// TIA Portal project "Project-Sticle" (V15.1)

(* hardware
DEVICE "S71500/ET200MP station_1"  S7-1500 station
   slot 0: "Rail_0"  Rack  6ES7 590-1***0-0AA0
   slot 1: "PLC_1"  CPU 1513-1 PN  6ES7 513-1AL02-0AB0  V2.6
      slot 3: "CPU display_1"  6ES7591-1AA00-0AA0
DEVICE "HMI_1"  KTP900 Basic PN
   slot 0: "HMI_1"  KTP900 Basic PN  6AV2 123-2JB03-0AX0  15.1.0.0
   slot 1: "HMI_RT_1"  KTP900 Basic PN  6AV2 123-2JB03-0AX0  15.1.0.0
   slot 5: "HMI_1.IE_CP_1"  PROFINET Interface  15.0.1.0
      slot 1: "PROFINET Interface_1"  PROFINET Interface
         slot 1: "Port_1"  Port
*)

// ===== PLC "PLC_1"  CPU 1513-1 PN =====

VAR_GLOBAL   // PLC tag table "Default tag table"
   "Clock_Byte" AT %MB0 : Byte;
   "Clock_10Hz" AT %M0.0 : Bool;
   "Clock_5Hz" AT %M0.1 : Bool;
   "Clock_2.5Hz" AT %M0.2 : Bool;
   "Clock_2Hz" AT %M0.3 : Bool;
   "Clock_1.25Hz" AT %M0.4 : Bool;
   "Clock_1Hz" AT %M0.5 : Bool;
   "Clock_0.625Hz" AT %M0.6 : Bool;
   "Clock_0.5Hz" AT %M0.7 : Bool;
END_VAR

DATA_BLOCK "Avarii"   // DB1
{ S7_Optimized_Access := 'TRUE' }
VERSION : 0.1
   VAR
      esd : Bool;
      esd_btn : Bool;
      reset_esd : Bool;
      confirmare_neprimita_actuator : Bool;
      reset_avarii : Bool;
      avarie_imbuteliere : Bool;
      avarie_capace : Bool;
      avarie_eticheta : Bool;
      avarie_impachetare : Bool;
      avarie_cuptor : Bool;
      avarie_generala : Bool;
      timer_confirmare : Time;
      timer_umplere : Time;
      timer_eticheta : Time;
      timer_capac : Time;
      timer_impachetare : Time;
      var_confirmare : Bool;
      timer_secunde_imbuteliere : Time;
      timer_secunde_confirmare : Time;
      timer_secunde_capac : Time;
      timer_secunde_impachetare : Time;
      timer_secunde_eticheta : Time;
      timer_cuptor : Time;
      timer_secunde_cutor : Time;
   END_VAR
BEGIN
END_DATA_BLOCK

DATA_BLOCK "Alarme"   // DB2
{ S7_Optimized_Access := 'TRUE' }
VERSION : 0.1
   VAR
      alarme_gather : Word;
      alarme_vect : Array[0..15] of Bool;
   END_VAR
BEGIN
END_DATA_BLOCK

DATA_BLOCK "Banda"   // DB4
{ S7_Optimized_Access := 'TRUE' }
VERSION : 0.1
   VAR
      banda_pornita_1 : Bool;
      prm_pornire_banda11 : Bool;
      prm_pornire_banda12 : Bool;
      banda_oprita_2 : Bool;
      banda_oprita_3 : Bool;
      banda_oprita_4 : Bool;
      banda_oprita_5 : Bool;
   END_VAR
BEGIN
END_DATA_BLOCK

DATA_BLOCK "Aparate"   // DB5
{ S7_Optimized_Access := 'TRUE' }
VERSION : 0.1
   VAR
      numar_sticle_cerut : UInt;
      numar_sticle_cerut_aux : UInt;
      numar_sticle : UInt;
      inchidere_actuator : Bool;
      deschidere_actuator : Bool;
      confirmare_actuator : Bool;
      timp_umplere_user : Time;
      timp_umplere_secunde : Time;
      terminat_imbuteliere : Bool;
      ajuns_capace : Bool;
      plecat_capace : Bool;
      ajuns_eticheta : Bool;
      plecat_ethicheta : Bool;
      ajuns_impachetare : Bool;
      plecat_impachetare : Bool;
      ajuns_cuptor : Bool;
      plecat_cuptor : Bool;
      nivel_palet : UInt;
      limita_palet : UInt;
      timp_cuptor : Time;
      timp_cuptor_secunde : Time;
   END_VAR
BEGIN
END_DATA_BLOCK

DATA_BLOCK "Butoane/Permisiuni"   // DB6
{ S7_Optimized_Access := 'TRUE' }
VERSION : 0.1
   VAR
      btn_start : Bool;
      permisiune_start : Bool;
      nr_sticle_complet : Bool;
      pauza : Bool;
   END_VAR
BEGIN
END_DATA_BLOCK

DATA_BLOCK "Rising_edges"   // DB7
{ S7_Optimized_Access := 'TRUE' }
VERSION : 0.1
   VAR
      re1 : Bool;
      re2 : Bool;
      re3 : Bool;
      re4 : Bool;
   END_VAR
BEGIN
END_DATA_BLOCK

DATA_BLOCK "Hysteresis_DB"   // DB15
{ S7_Optimized_Access := 'TRUE' }
VERSION : 0.1
// stored: InstanceOfName Hysteresis
"Hysteresis"
BEGIN
END_DATA_BLOCK

DATA_BLOCK "Variabile_Hysteresis"   // DB16
{ S7_Optimized_Access := 'TRUE' }
VERSION : 0.1
   VAR
      bool_cond : Bool;
      Hy_val : Real;
      Setpoint : Real;
      temp : Real;
      lim_inf : Real;
      lim_sup : Real;
      limita_inf_pt_timer : Real;
      dif_lim_inf : Real;
   END_VAR
BEGIN
END_DATA_BLOCK

DATA_BLOCK "Turn_vizual"   // DB17
{ S7_Optimized_Access := 'TRUE' }
VERSION : 0.1
   VAR
      led_rosu : Bool;
      led_verde : Bool;
      led_galben : Bool;
   END_VAR
BEGIN
END_DATA_BLOCK

DATA_BLOCK "Brat_descarcare_DB"   // DB18
{ S7_Optimized_Access := 'TRUE' }
VERSION : 0.1
// stored: InstanceOfName Brat_descarcare
"Brat_descarcare"
BEGIN
END_DATA_BLOCK

DATA_BLOCK "Stari_brat_descarcare"   // DB19
{ S7_Optimized_Access := 'TRUE' }
VERSION : 0.1
   VAR
      ready : Bool;
      finish : Bool;
      running : Bool;
   END_VAR
BEGIN
END_DATA_BLOCK

DATA_BLOCK "Cuastom 0,2HZ clock_DB"   // DB20
{ S7_Optimized_Access := 'TRUE' }
VERSION : 0.1
// stored: InstanceOfName Custom 0,2HZ clock
"Custom 0,2HZ clock"
BEGIN
END_DATA_BLOCK

DATA_BLOCK "Cuptor_DB"   // DB21
{ S7_Optimized_Access := 'TRUE' }
VERSION : 0.1
// stored: InstanceOfName Cuptor
"Cuptor"
BEGIN
END_DATA_BLOCK

// folder: System blocks/Program resources

DATA_BLOCK "timer_confirmare_actuator"   // DB8
{ S7_Optimized_Access := 'TRUE' }
AUTHOR : Simatic
FAMILY : IEC
NAME : IEC_TMR
VERSION : 1.0
// stored: InstanceOfName IEC_TIMER
"IEC_TIMER"
BEGIN
END_DATA_BLOCK

DATA_BLOCK "timer_imbuteliere"   // DB9
{ S7_Optimized_Access := 'TRUE' }
AUTHOR : Simatic
FAMILY : IEC
NAME : IEC_TMR
VERSION : 1.0
// stored: InstanceOfName IEC_TIMER
"IEC_TIMER"
BEGIN
END_DATA_BLOCK

DATA_BLOCK "timer_reset_btn_avarii"   // DB10
{ S7_Optimized_Access := 'TRUE' }
AUTHOR : Simatic
FAMILY : IEC
NAME : IEC_TMR
VERSION : 1.0
// stored: InstanceOfName IEC_TIMER
"IEC_TIMER"
BEGIN
END_DATA_BLOCK

DATA_BLOCK "timer_capace"   // DB11
{ S7_Optimized_Access := 'TRUE' }
AUTHOR : Simatic
FAMILY : IEC
NAME : IEC_TMR
VERSION : 1.0
// stored: InstanceOfName IEC_TIMER
"IEC_TIMER"
BEGIN
END_DATA_BLOCK

DATA_BLOCK "timer_eticheta"   // DB12
{ S7_Optimized_Access := 'TRUE' }
AUTHOR : Simatic
FAMILY : IEC
NAME : IEC_TMR
VERSION : 1.0
// stored: InstanceOfName IEC_TIMER
"IEC_TIMER"
BEGIN
END_DATA_BLOCK

DATA_BLOCK "timer_impachetare"   // DB13
{ S7_Optimized_Access := 'TRUE' }
AUTHOR : Simatic
FAMILY : IEC
NAME : IEC_TMR
VERSION : 1.0
// stored: InstanceOfName IEC_TIMER
"IEC_TIMER"
BEGIN
END_DATA_BLOCK

DATA_BLOCK "reset_esd"   // DB14
{ S7_Optimized_Access := 'TRUE' }
AUTHOR : Simatic
FAMILY : IEC
NAME : IEC_TMR
VERSION : 1.0
// stored: InstanceOfName IEC_TIMER
"IEC_TIMER"
BEGIN
END_DATA_BLOCK

// folder: (top level)

FUNCTION_BLOCK "Hysteresis"   // FB1, LAD
{ S7_Optimized_Access := 'TRUE' }
VERSION : 0.1
   VAR_INPUT
      HY_val : Real;
      Setpoint : Real;
   END_VAR
   VAR_OUTPUT
      h_lim_sup : Real;
      h_lim_inf : Real;
      bool_cond : Bool;
   END_VAR
   VAR_IN_OUT
      temp : Real;
   END_VAR
   VAR
      re1 : Bool;
      re2 : Bool;
      urcare : Bool;
   END_VAR
   VAR_TEMP   // added for the SCL form of the ladder/FBD networks
      _w1 : Bool;
   END_VAR
BEGIN

REGION Network 1: daca are comanda de bool, sa creasca
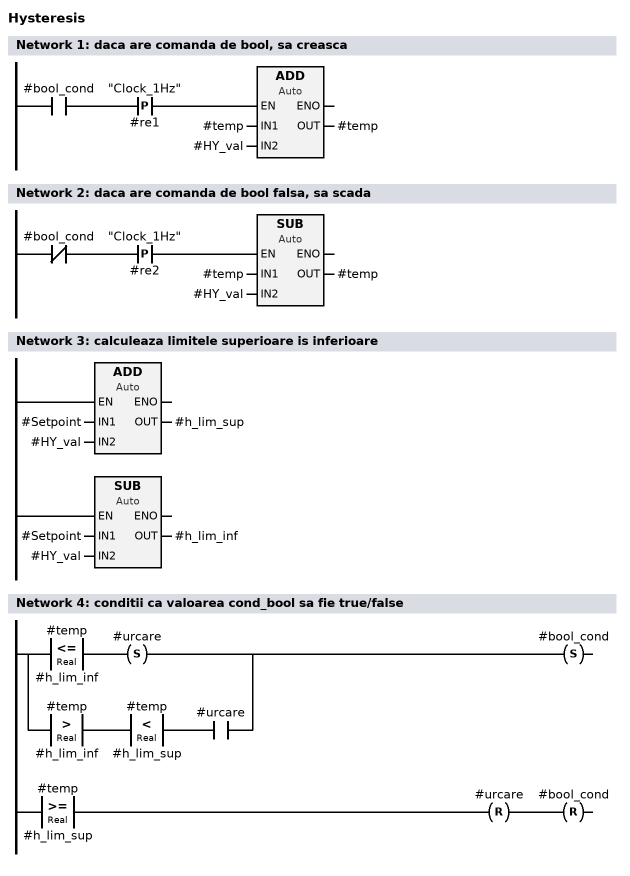
   RUNG wire#powerrail
      Contact( #bool_cond )
      P_Contact(operand := "Clock_1Hz", bit := #re1)
      Add(in1 := #temp, in2 := #HY_val, out => #temp)
   END_RUNG
   // the same network as SCL:
   #_w1 := #bool_cond AND "Clock_1Hz" AND NOT #re1;   // rising edge of "Clock_1Hz"
   #re1 := "Clock_1Hz";
   IF #_w1 THEN #temp := #temp + #HY_val; END_IF;
END_REGION

REGION Network 2: daca are comanda de bool falsa, sa scada
   RUNG wire#powerrail
      I_Contact( #bool_cond )
      P_Contact(operand := "Clock_1Hz", bit := #re2)
      Sub(in1 := #temp, in2 := #HY_val, out => #temp)
   END_RUNG
   // the same network as SCL:
   #_w1 := NOT #bool_cond AND "Clock_1Hz" AND NOT #re2;   // rising edge of "Clock_1Hz"
   #re2 := "Clock_1Hz";
   IF #_w1 THEN #temp := #temp - #HY_val; END_IF;
END_REGION

REGION Network 3: calculeaza limitele superioare is inferioare
   RUNG wire#powerrail
      Add(in1 := #Setpoint, in2 := #HY_val, out => #h_lim_sup)
   END_RUNG
   RUNG wire#powerrail
      Sub(in1 := #Setpoint, in2 := #HY_val, out => #h_lim_inf)
   END_RUNG
   // the same network as SCL:
   #h_lim_sup := #Setpoint + #HY_val;
   #h_lim_inf := #Setpoint - #HY_val;
END_REGION

REGION Network 4: conditii ca valoarea cond_bool sa fie true/false
   RUNG wire#powerrail
      { S7_Templates := "SrcType := Real" } LE_Contact(in1 := #temp, in2 := #h_lim_inf)
      S_Coil( #urcare )
      wire#w1
      S_Coil( #bool_cond )
   END_RUNG
   RUNG wire#powerrail
      { S7_Templates := "SrcType := Real" } GT_Contact(in1 := #temp, in2 := #h_lim_inf)
      { S7_Templates := "SrcType := Real" } LT_Contact(in1 := #temp, in2 := #h_lim_sup)
      Contact( #urcare )
   END_RUNG wire#w1
   RUNG wire#powerrail
      { S7_Templates := "SrcType := Real" } GE_Contact(in1 := #temp, in2 := #h_lim_sup)
      R_Coil( #urcare )
      R_Coil( #bool_cond )
   END_RUNG
   // the same network as SCL:
   #_w1 := #temp <= #h_lim_inf;
   IF #_w1 THEN #urcare := TRUE; END_IF;
   IF #_w1 OR ((#temp > #h_lim_inf) AND (#temp < #h_lim_sup) AND #urcare) THEN #bool_cond := TRUE; END_IF;
   IF #temp >= #h_lim_sup THEN
       #urcare := FALSE;
       #bool_cond := FALSE;
   END_IF;
END_REGION
END_FUNCTION_BLOCK

FUNCTION_BLOCK "Brat_descarcare"   // FB2, LAD
{ S7_Optimized_Access := 'TRUE' }
VERSION : 0.1
   VAR_OUTPUT
      ready : Bool;
      finish : Bool;
      running : Bool;
   END_VAR
   VAR_IN_OUT
      permisiune : Bool;
      nivel_palet : UInt;
   END_VAR
   VAR
      re1 : Bool;
      counter_custom_clock : UInt;
      "bool value" : Bool;
   END_VAR
   VAR_TEMP   // added for the SCL form of the ladder/FBD networks
      _w1 : Bool;
   END_VAR
BEGIN

REGION Network 1: daca e ready si are permisiune, sa treaca pe run
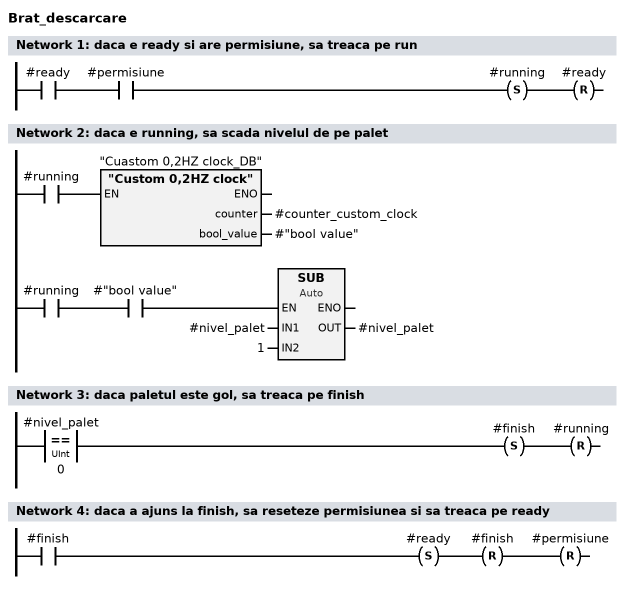
   RUNG wire#powerrail
      Contact( #ready )
      Contact( #permisiune )
      S_Coil( #running )
      R_Coil( #ready )
   END_RUNG
   // the same network as SCL:
   IF #ready AND #permisiune THEN
       #running := TRUE;
       #ready := FALSE;
   END_IF;
END_REGION

REGION Network 2: daca e running, sa scada nivelul de pe palet
   RUNG wire#powerrail
      Contact( #running )
      "Cuastom 0,2HZ clock_DB"("counter" => #counter_custom_clock, bool_value => #"bool value")
   END_RUNG
   RUNG wire#powerrail
      Contact( #running )
      Contact( #"bool value" )
      Sub(in1 := #nivel_palet, in2 := 1, out => #nivel_palet)
   END_RUNG
   // the same network as SCL:
   IF #running THEN
       "Cuastom 0,2HZ clock_DB"("counter" => #counter_custom_clock, bool_value => #"bool value");   // "Custom 0,2HZ clock"
   END_IF;
   IF #running AND #"bool value" THEN #nivel_palet := #nivel_palet - 1; END_IF;
END_REGION

REGION Network 3: daca paletul este gol, sa treaca pe finish
   RUNG wire#powerrail
      { S7_Templates := "SrcType := UInt" } EQ_Contact(in1 := #nivel_palet, in2 := 0)
      S_Coil( #finish )
      R_Coil( #running )
   END_RUNG
   // the same network as SCL:
   IF #nivel_palet = 0 THEN
       #finish := TRUE;
       #running := FALSE;
   END_IF;
END_REGION

REGION Network 4: daca a ajuns la finish, sa reseteze permisiunea si sa treaca pe ready
   RUNG wire#powerrail
      Contact( #finish )
      S_Coil( #ready )
      R_Coil( #finish )
      R_Coil( #permisiune )
   END_RUNG
   // the same network as SCL:
   IF #finish THEN #ready := TRUE; END_IF;
   #_w1 := #finish;
   IF #_w1 THEN
       #finish := FALSE;
       #permisiune := FALSE;
   END_IF;
END_REGION
END_FUNCTION_BLOCK

FUNCTION_BLOCK "Custom 0,2HZ clock"   // FB3, LAD
{ S7_Optimized_Access := 'TRUE' }
VERSION : 0.1
   VAR_OUTPUT
      "counter" : UInt;
      bool_value : Bool;
   END_VAR
   VAR
      re : Bool;
   END_VAR
   VAR_TEMP   // added for the SCL form of the ladder/FBD networks
      _w1 : Bool;
   END_VAR
BEGIN

REGION Network 1: adauga la counter
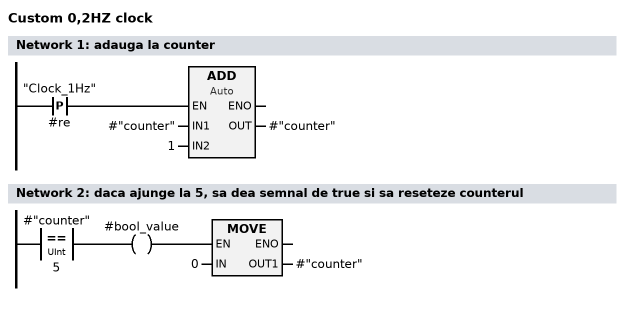
   RUNG wire#powerrail
      P_Contact(operand := "Clock_1Hz", bit := #re)
      Add(in1 := #"counter", in2 := 1, out => #"counter")
   END_RUNG
   // the same network as SCL:
   #_w1 := "Clock_1Hz" AND NOT #re;   // rising edge of "Clock_1Hz"
   #re := "Clock_1Hz";
   IF #_w1 THEN #"counter" := #"counter" + 1; END_IF;
END_REGION

REGION Network 2: daca ajunge la 5, sa dea semnal de true si sa reseteze counterul
   RUNG wire#powerrail
      { S7_Templates := "SrcType := UInt" } EQ_Contact(in1 := #"counter", in2 := 5)
      Coil( #bool_value )
      Move(in := 0, out1 => #"counter")
   END_RUNG
   // the same network as SCL:
   #bool_value := #"counter" = 5;
   IF #bool_value THEN #"counter" := 0; END_IF;
END_REGION
END_FUNCTION_BLOCK

FUNCTION_BLOCK "Cuptor"   // FB4, LAD
{ S7_Optimized_Access := 'TRUE' }
VERSION : 0.1
   VAR_INPUT
      hysteresis_setpoint : Real;
      dif_lim_inf : Real;
      timp_cuptor : Time;
      buton_perm_start : Bool;
      banda_oprita : Bool;
      pauza : Bool;
      avarie_generala : Bool;
      esd : Bool;
   END_VAR
   VAR_OUTPUT
      timer_cuptor_out : Time;
   END_VAR
   VAR_IN_OUT
      b_oprita : Bool;
      plecat_cuptor : Bool;
      ajuns_cuptor : Bool;
      hy_bool_cond : Bool;
      timp_cuptor_sec : Time;
      lim_inf_pt_timer : Real;
      temp : Real;
      hy_val : Real;
      lim_sup : Real;
      lim_inf : Real;
   END_VAR
   VAR
      timer_cuptor : TON_TIME;
   END_VAR
BEGIN

REGION Network 1: calculeaza limita inferioara pt timer la cuptor si timpul in secunde la cuptor
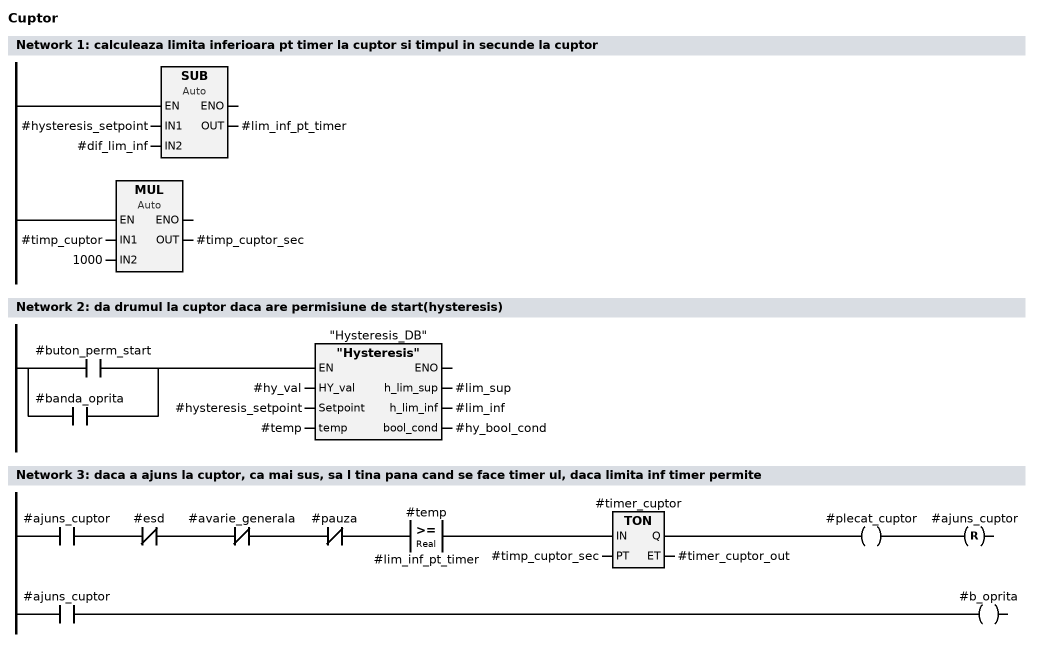
   RUNG wire#powerrail
      Sub(in1 := #hysteresis_setpoint, in2 := #dif_lim_inf, out => #lim_inf_pt_timer)
   END_RUNG
   RUNG wire#powerrail
      Mul(in1 := #timp_cuptor, in2 := 1000, out => #timp_cuptor_sec)
   END_RUNG
   // the same network as SCL:
   #lim_inf_pt_timer := #hysteresis_setpoint - #dif_lim_inf;
   #timp_cuptor_sec := #timp_cuptor * 1000;
END_REGION

REGION Network 2: da drumul la cuptor daca are permisiune de start(hysteresis)
   RUNG wire#powerrail
      Contact( #buton_perm_start )
      wire#w1
      "Hysteresis_DB"(HY_val := #hy_val, Setpoint := #hysteresis_setpoint, temp := #temp, h_lim_sup => #lim_sup, h_lim_inf => #lim_inf, bool_cond => #hy_bool_cond)
   END_RUNG
   RUNG wire#powerrail
      Contact( #banda_oprita )
   END_RUNG wire#w1
   // the same network as SCL:
   IF #buton_perm_start OR #banda_oprita THEN
       "Hysteresis_DB"(HY_val := #hy_val,   // "Hysteresis"
                       Setpoint := #hysteresis_setpoint,
                       temp := #temp,
                       h_lim_sup => #lim_sup,
                       h_lim_inf => #lim_inf,
                       bool_cond => #hy_bool_cond);
   END_IF;
END_REGION

REGION Network 3: daca a ajuns la cuptor, ca mai sus, sa l tina pana cand se face timer ul, daca limita inf timer permite
   #timer_cuptor(IN := #ajuns_cuptor AND NOT #esd AND NOT #avarie_generala AND NOT #pauza AND (#temp >= #lim_inf_pt_timer),   // TON
                 PT := #timp_cuptor_sec,
                 ET => #timer_cuptor_out);
   #plecat_cuptor := #timer_cuptor.Q;
   IF #timer_cuptor.Q THEN #ajuns_cuptor := FALSE; END_IF;
   #b_oprita := #ajuns_cuptor;
END_REGION
END_FUNCTION_BLOCK

ORGANIZATION_BLOCK "Main"   // OB1, LAD, ProgramCycle
TITLE = "Main Program Sweep (Cycle)"
{ S7_Optimized_Access := 'TRUE' }
VERSION : 0.1
   VAR_INPUT
      Initial_Call : Bool;   // Initial call of this OB
      Remanence : Bool;   // =True, if remanent data are available
   END_VAR
   VAR_TEMP   // added for the SCL form of the ladder/FBD networks
      _w1 : Bool;
   END_VAR
BEGIN

REGION Network 1: permisiune start(adauga la final si avarie generala pt fiecare aparat in parte)
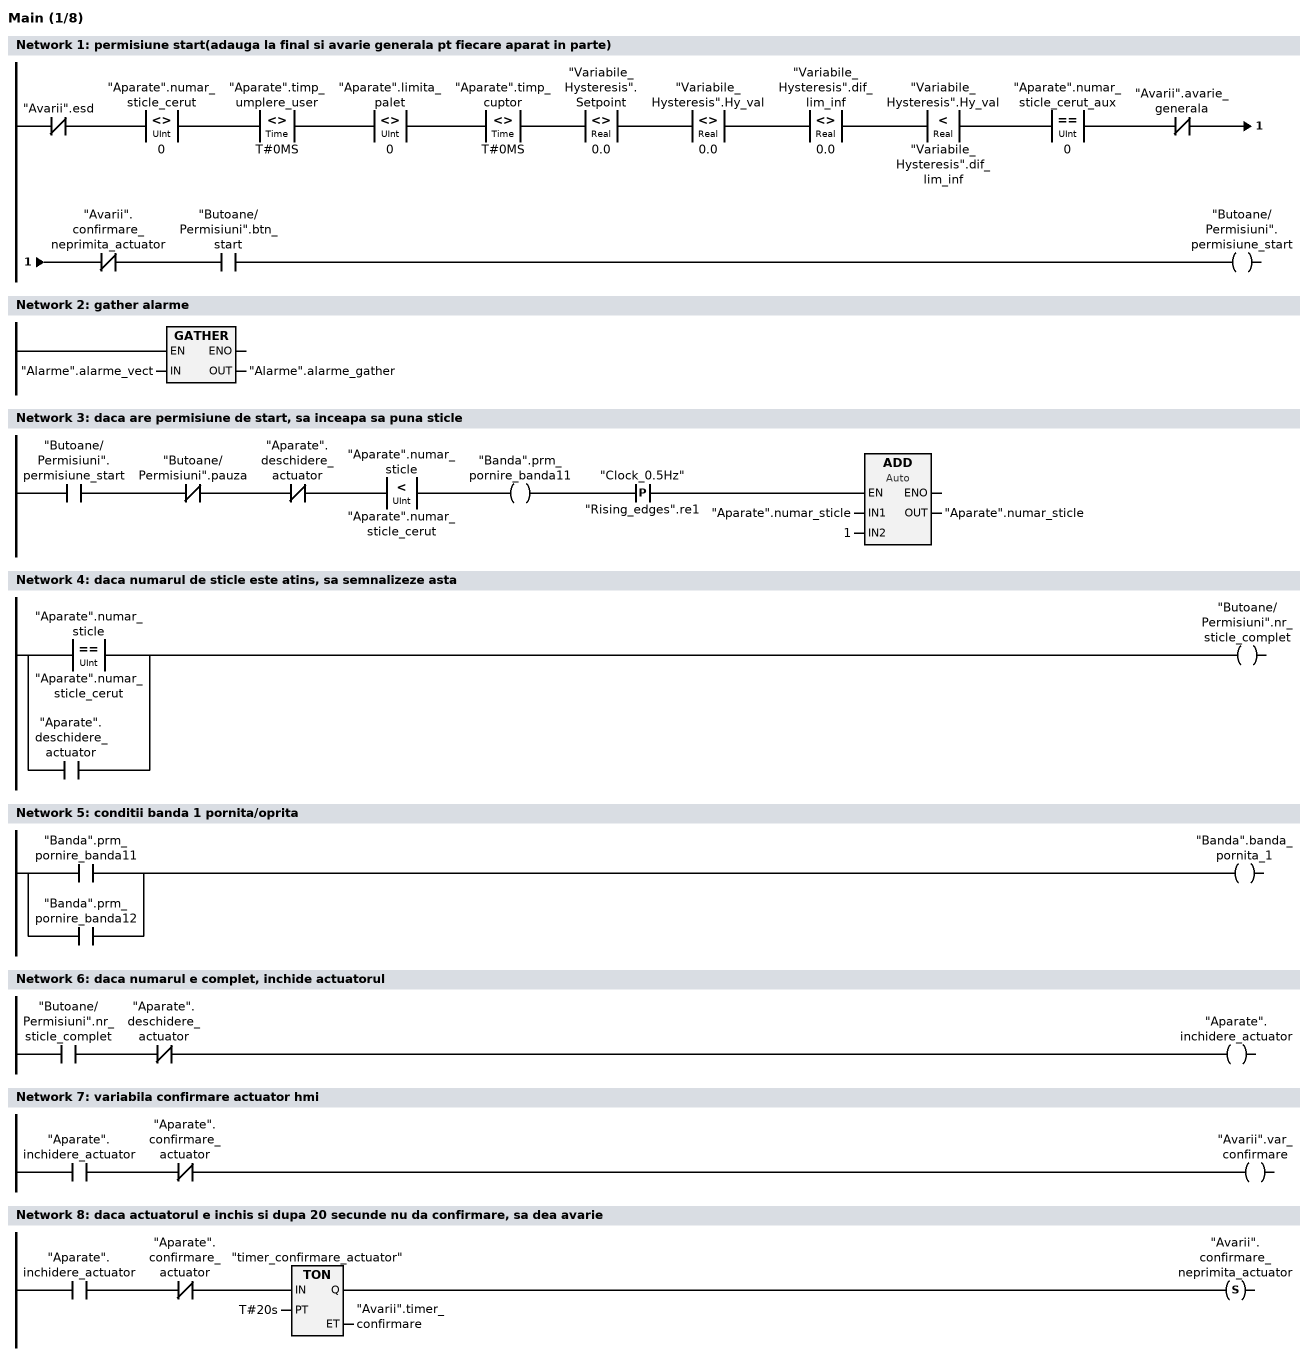
   RUNG wire#powerrail
      I_Contact( "Avarii".esd )
      { S7_Templates := "SrcType := UInt" } NE_Contact(in1 := "Aparate".numar_sticle_cerut, in2 := 0)
      { S7_Templates := "SrcType := Time" } NE_Contact(in1 := "Aparate".timp_umplere_user, in2 := T#0MS)
      { S7_Templates := "SrcType := UInt" } NE_Contact(in1 := "Aparate".limita_palet, in2 := 0)
      { S7_Templates := "SrcType := Time" } NE_Contact(in1 := "Aparate".timp_cuptor, in2 := T#0MS)
      { S7_Templates := "SrcType := Real" } NE_Contact(in1 := "Variabile_Hysteresis".Setpoint, in2 := 0.0)
      { S7_Templates := "SrcType := Real" } NE_Contact(in1 := "Variabile_Hysteresis".Hy_val, in2 := 0.0)
      { S7_Templates := "SrcType := Real" } NE_Contact(in1 := "Variabile_Hysteresis".dif_lim_inf, in2 := 0.0)
      { S7_Templates := "SrcType := Real" } LT_Contact(in1 := "Variabile_Hysteresis".Hy_val, in2 := "Variabile_Hysteresis".dif_lim_inf)
      { S7_Templates := "SrcType := UInt" } EQ_Contact(in1 := "Aparate".numar_sticle_cerut_aux, in2 := 0)
      I_Contact( "Avarii".avarie_generala )
      I_Contact( "Avarii".confirmare_neprimita_actuator )
      Contact( "Butoane/Permisiuni".btn_start )
      Coil( "Butoane/Permisiuni".permisiune_start )
   END_RUNG
   // the same network as SCL:
   "Butoane/Permisiuni".permisiune_start := NOT "Avarii".esd AND ("Aparate".numar_sticle_cerut <> 0) AND ("Aparate".timp_umplere_user <> T#0MS) AND ("Aparate".limita_palet <> 0) AND ("Aparate".timp_cuptor <> T#0MS) AND ("Variabile_Hysteresis".Setpoint <> 0.0) AND ("Variabile_Hysteresis".Hy_val <> 0.0) AND ("Variabile_Hysteresis".dif_lim_inf <> 0.0) AND ("Variabile_Hysteresis".Hy_val < "Variabile_Hysteresis".dif_lim_inf) AND ("Aparate".numar_sticle_cerut_aux = 0) AND NOT "Avarii".avarie_generala AND NOT "Avarii".confirmare_neprimita_actuator AND "Butoane/Permisiuni".btn_start;
END_REGION

REGION Network 2: gather alarme
   GATHER(IN := "Alarme".alarme_vect, OUT => "Alarme".alarme_gather);
END_REGION

REGION Network 3: daca are permisiune de start, sa inceapa sa puna sticle
   RUNG wire#powerrail
      Contact( "Butoane/Permisiuni".permisiune_start )
      I_Contact( "Butoane/Permisiuni".pauza )
      I_Contact( "Aparate".deschidere_actuator )
      { S7_Templates := "SrcType := UInt" } LT_Contact(in1 := "Aparate".numar_sticle, in2 := "Aparate".numar_sticle_cerut)
      Coil( "Banda".prm_pornire_banda11 )
      P_Contact(operand := "Clock_0.5Hz", bit := "Rising_edges".re1)
      Add(in1 := "Aparate".numar_sticle, in2 := 1, out => "Aparate".numar_sticle)
   END_RUNG
   // the same network as SCL:
   "Banda".prm_pornire_banda11 := "Butoane/Permisiuni".permisiune_start AND NOT "Butoane/Permisiuni".pauza AND NOT "Aparate".deschidere_actuator AND ("Aparate".numar_sticle < "Aparate".numar_sticle_cerut);
   #_w1 := "Banda".prm_pornire_banda11 AND "Clock_0.5Hz" AND NOT "Rising_edges".re1;   // rising edge of "Clock_0.5Hz"
   "Rising_edges".re1 := "Clock_0.5Hz";
   IF #_w1 THEN "Aparate".numar_sticle := "Aparate".numar_sticle + 1; END_IF;
END_REGION

REGION Network 4: daca numarul de sticle este atins, sa semnalizeze asta
   RUNG wire#powerrail
      { S7_Templates := "SrcType := UInt" } EQ_Contact(in1 := "Aparate".numar_sticle, in2 := "Aparate".numar_sticle_cerut)
      wire#w1
      Coil( "Butoane/Permisiuni".nr_sticle_complet )
   END_RUNG
   RUNG wire#powerrail
      Contact( "Aparate".deschidere_actuator )
   END_RUNG wire#w1
   // the same network as SCL:
   "Butoane/Permisiuni".nr_sticle_complet := ("Aparate".numar_sticle = "Aparate".numar_sticle_cerut) OR "Aparate".deschidere_actuator;
END_REGION

REGION Network 5: conditii banda 1 pornita/oprita
   RUNG wire#powerrail
      Contact( "Banda".prm_pornire_banda11 )
      wire#w1
      Coil( "Banda".banda_pornita_1 )
   END_RUNG
   RUNG wire#powerrail
      Contact( "Banda".prm_pornire_banda12 )
   END_RUNG wire#w1
   // the same network as SCL:
   "Banda".banda_pornita_1 := "Banda".prm_pornire_banda11 OR "Banda".prm_pornire_banda12;
END_REGION

REGION Network 6: daca numarul e complet, inchide actuatorul
   RUNG wire#powerrail
      Contact( "Butoane/Permisiuni".nr_sticle_complet )
      I_Contact( "Aparate".deschidere_actuator )
      Coil( "Aparate".inchidere_actuator )
   END_RUNG
   // the same network as SCL:
   "Aparate".inchidere_actuator := "Butoane/Permisiuni".nr_sticle_complet AND NOT "Aparate".deschidere_actuator;
END_REGION

REGION Network 7: variabila confirmare actuator hmi
   RUNG wire#powerrail
      Contact( "Aparate".inchidere_actuator )
      I_Contact( "Aparate".confirmare_actuator )
      Coil( "Avarii".var_confirmare )
   END_RUNG
   // the same network as SCL:
   "Avarii".var_confirmare := "Aparate".inchidere_actuator AND NOT "Aparate".confirmare_actuator;
END_REGION

REGION Network 8: daca actuatorul e inchis si dupa 20 secunde nu da confirmare, sa dea avarie
   "timer_confirmare_actuator".TON(IN := "Aparate".inchidere_actuator AND NOT "Aparate".confirmare_actuator,
                           PT := T#20s,
                           ET => "Avarii".timer_confirmare);
   IF "timer_confirmare_actuator".Q THEN "Avarii".confirmare_neprimita_actuator := TRUE; END_IF;
END_REGION

REGION Network 9: daca nr de sticle curent nu este cat cel cerut, sa nu poata sa dea confirmarea actuatorului
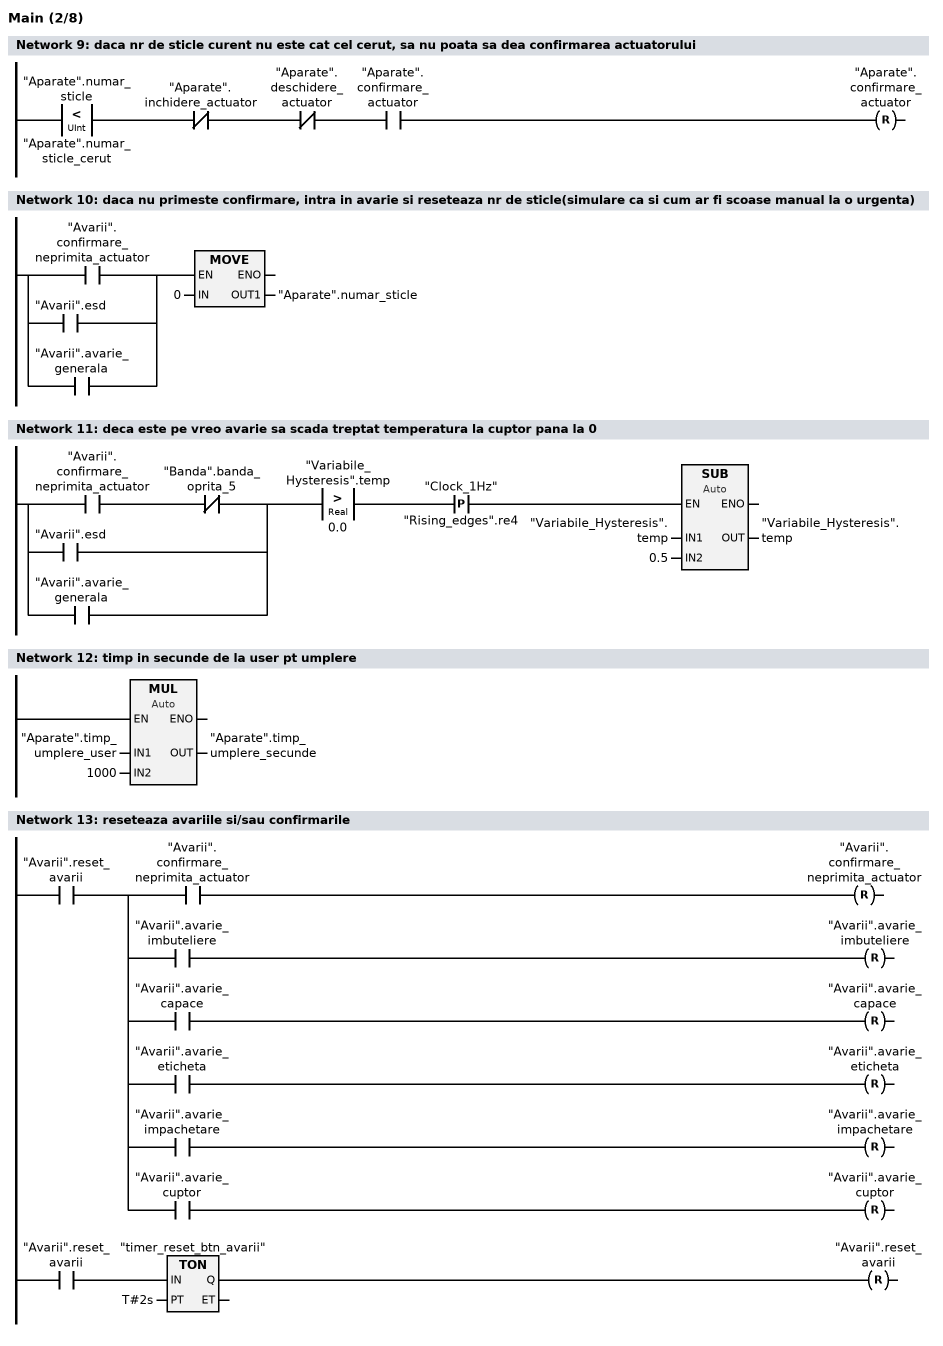
   RUNG wire#powerrail
      { S7_Templates := "SrcType := UInt" } LT_Contact(in1 := "Aparate".numar_sticle, in2 := "Aparate".numar_sticle_cerut)
      I_Contact( "Aparate".inchidere_actuator )
      I_Contact( "Aparate".deschidere_actuator )
      Contact( "Aparate".confirmare_actuator )
      R_Coil( "Aparate".confirmare_actuator )
   END_RUNG
   // the same network as SCL:
   IF ("Aparate".numar_sticle < "Aparate".numar_sticle_cerut) AND NOT "Aparate".inchidere_actuator AND NOT "Aparate".deschidere_actuator AND "Aparate".confirmare_actuator THEN
       "Aparate".confirmare_actuator := FALSE;
   END_IF;
END_REGION

REGION Network 10: daca nu primeste confirmare, intra in avarie si reseteaza nr de sticle(simulare ca si cum ar fi scoase manual la o urgenta)
   RUNG wire#powerrail
      Contact( "Avarii".confirmare_neprimita_actuator )
      wire#w1
      Move(in := 0, out1 => "Aparate".numar_sticle)
   END_RUNG
   RUNG wire#powerrail
      Contact( "Avarii".esd )
   END_RUNG wire#w1
   RUNG wire#powerrail
      Contact( "Avarii".avarie_generala )
   END_RUNG wire#w1
   // the same network as SCL:
   IF "Avarii".confirmare_neprimita_actuator OR "Avarii".esd OR "Avarii".avarie_generala THEN
       "Aparate".numar_sticle := 0;
   END_IF;
END_REGION

REGION Network 11: deca este pe vreo avarie sa scada treptat temperatura la cuptor pana la 0
   RUNG wire#powerrail
      Contact( "Avarii".confirmare_neprimita_actuator )
      I_Contact( "Banda".banda_oprita_5 )
      wire#w1
      { S7_Templates := "SrcType := Real" } GT_Contact(in1 := "Variabile_Hysteresis".temp, in2 := 0.0)
      P_Contact(operand := "Clock_1Hz", bit := "Rising_edges".re4)
      Sub(in1 := "Variabile_Hysteresis".temp, in2 := 0.5, out => "Variabile_Hysteresis".temp)
   END_RUNG
   RUNG wire#powerrail
      Contact( "Avarii".esd )
   END_RUNG wire#w1
   RUNG wire#powerrail
      Contact( "Avarii".avarie_generala )
   END_RUNG wire#w1
   // the same network as SCL:
   #_w1 := (("Avarii".confirmare_neprimita_actuator AND NOT "Banda".banda_oprita_5) OR "Avarii".esd OR "Avarii".avarie_generala) AND ("Variabile_Hysteresis".temp > 0.0) AND "Clock_1Hz" AND NOT "Rising_edges".re4;   // rising edge of "Clock_1Hz"
   "Rising_edges".re4 := "Clock_1Hz";
   IF #_w1 THEN "Variabile_Hysteresis".temp := "Variabile_Hysteresis".temp - 0.5; END_IF;
END_REGION

REGION Network 12: timp in secunde de la user pt umplere
   RUNG wire#powerrail
      Mul(in1 := "Aparate".timp_umplere_user, in2 := 1000, out => "Aparate".timp_umplere_secunde)
   END_RUNG
   // the same network as SCL:
   "Aparate".timp_umplere_secunde := "Aparate".timp_umplere_user * 1000;
END_REGION

REGION Network 13: reseteaza avariile si/sau confirmarile
   IF "Avarii".reset_avarii AND "Avarii".confirmare_neprimita_actuator THEN
       "Avarii".confirmare_neprimita_actuator := FALSE;
   END_IF;
   IF "Avarii".reset_avarii AND "Avarii".avarie_imbuteliere THEN
       "Avarii".avarie_imbuteliere := FALSE;
   END_IF;
   IF "Avarii".reset_avarii AND "Avarii".avarie_capace THEN "Avarii".avarie_capace := FALSE; END_IF;
   IF "Avarii".reset_avarii AND "Avarii".avarie_eticheta THEN "Avarii".avarie_eticheta := FALSE; END_IF;
   IF "Avarii".reset_avarii AND "Avarii".avarie_impachetare THEN
       "Avarii".avarie_impachetare := FALSE;
   END_IF;
   IF "Avarii".reset_avarii AND "Avarii".avarie_cuptor THEN "Avarii".avarie_cuptor := FALSE; END_IF;
   "timer_reset_btn_avarii".TON(IN := "Avarii".reset_avarii, PT := T#2s);
   IF "timer_reset_btn_avarii".Q THEN "Avarii".reset_avarii := FALSE; END_IF;
END_REGION

REGION Network 14: reseteaza butonul de start in caz de esd/avarie
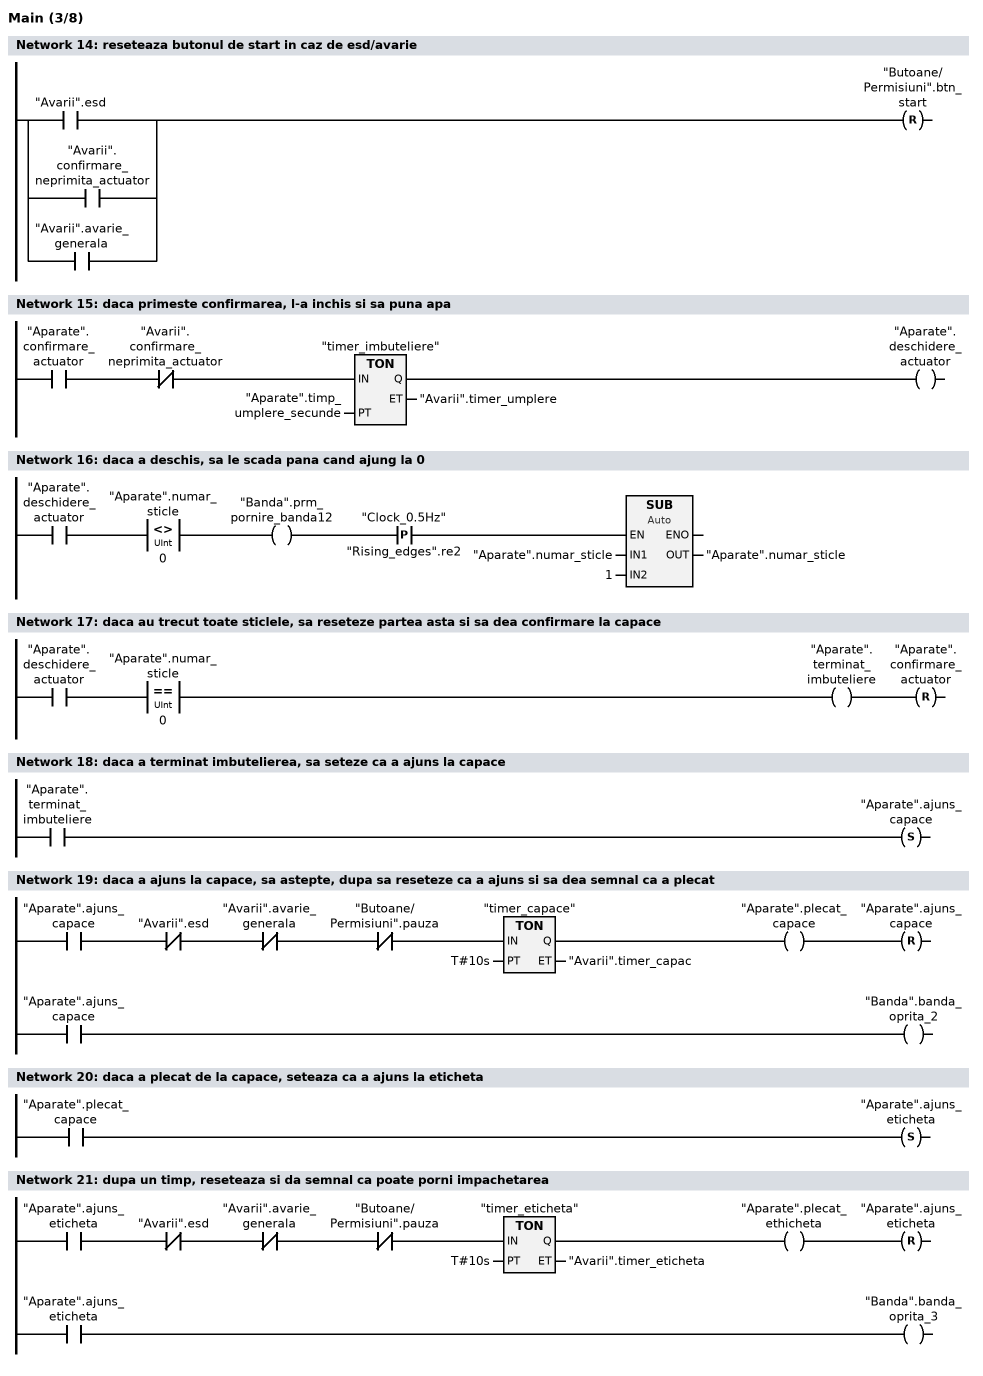
   RUNG wire#powerrail
      Contact( "Avarii".esd )
      wire#w1
      R_Coil( "Butoane/Permisiuni".btn_start )
   END_RUNG
   RUNG wire#powerrail
      Contact( "Avarii".confirmare_neprimita_actuator )
   END_RUNG wire#w1
   RUNG wire#powerrail
      Contact( "Avarii".avarie_generala )
   END_RUNG wire#w1
   // the same network as SCL:
   IF "Avarii".esd OR "Avarii".confirmare_neprimita_actuator OR "Avarii".avarie_generala THEN
       "Butoane/Permisiuni".btn_start := FALSE;
   END_IF;
END_REGION

REGION Network 15: daca primeste confirmarea, l-a inchis si sa puna apa
   "timer_imbuteliere".TON(IN := "Aparate".confirmare_actuator AND NOT "Avarii".confirmare_neprimita_actuator,
                           PT := "Aparate".timp_umplere_secunde,
                           ET => "Avarii".timer_umplere);
   "Aparate".deschidere_actuator := "timer_imbuteliere".Q;
END_REGION

REGION Network 16: daca a deschis, sa le scada pana cand ajung la 0
   RUNG wire#powerrail
      Contact( "Aparate".deschidere_actuator )
      { S7_Templates := "SrcType := UInt" } NE_Contact(in1 := "Aparate".numar_sticle, in2 := 0)
      Coil( "Banda".prm_pornire_banda12 )
      P_Contact(operand := "Clock_0.5Hz", bit := "Rising_edges".re2)
      Sub(in1 := "Aparate".numar_sticle, in2 := 1, out => "Aparate".numar_sticle)
   END_RUNG
   // the same network as SCL:
   "Banda".prm_pornire_banda12 := "Aparate".deschidere_actuator AND ("Aparate".numar_sticle <> 0);
   #_w1 := "Banda".prm_pornire_banda12 AND "Clock_0.5Hz" AND NOT "Rising_edges".re2;   // rising edge of "Clock_0.5Hz"
   "Rising_edges".re2 := "Clock_0.5Hz";
   IF #_w1 THEN "Aparate".numar_sticle := "Aparate".numar_sticle - 1; END_IF;
END_REGION

REGION Network 17: daca au trecut toate sticlele, sa reseteze partea asta si sa dea confirmare la capace
   RUNG wire#powerrail
      Contact( "Aparate".deschidere_actuator )
      { S7_Templates := "SrcType := UInt" } EQ_Contact(in1 := "Aparate".numar_sticle, in2 := 0)
      Coil( "Aparate".terminat_imbuteliere )
      R_Coil( "Aparate".confirmare_actuator )
   END_RUNG
   // the same network as SCL:
   "Aparate".terminat_imbuteliere := "Aparate".deschidere_actuator AND ("Aparate".numar_sticle = 0);
   IF "Aparate".terminat_imbuteliere THEN "Aparate".confirmare_actuator := FALSE; END_IF;
END_REGION

REGION Network 18: daca a terminat imbutelierea, sa seteze ca a ajuns la capace
   RUNG wire#powerrail
      Contact( "Aparate".terminat_imbuteliere )
      S_Coil( "Aparate".ajuns_capace )
   END_RUNG
   // the same network as SCL:
   IF "Aparate".terminat_imbuteliere THEN "Aparate".ajuns_capace := TRUE; END_IF;
END_REGION

REGION Network 19: daca a ajuns la capace, sa astepte, dupa sa reseteze ca a ajuns si sa dea semnal ca a plecat
   "timer_capace".TON(IN := "Aparate".ajuns_capace AND NOT "Avarii".esd AND NOT "Avarii".avarie_generala AND NOT "Butoane/Permisiuni".pauza,
                      PT := T#10s,
                      ET => "Avarii".timer_capac);
   "Aparate".plecat_capace := "timer_capace".Q;
   IF "timer_capace".Q THEN "Aparate".ajuns_capace := FALSE; END_IF;
   "Banda".banda_oprita_2 := "Aparate".ajuns_capace;
END_REGION

REGION Network 20: daca a plecat de la capace, seteaza ca a ajuns la eticheta
   RUNG wire#powerrail
      Contact( "Aparate".plecat_capace )
      S_Coil( "Aparate".ajuns_eticheta )
   END_RUNG
   // the same network as SCL:
   IF "Aparate".plecat_capace THEN "Aparate".ajuns_eticheta := TRUE; END_IF;
END_REGION

REGION Network 21: dupa un timp, reseteaza si da semnal ca poate porni impachetarea
   "timer_eticheta".TON(IN := "Aparate".ajuns_eticheta AND NOT "Avarii".esd AND NOT "Avarii".avarie_generala AND NOT "Butoane/Permisiuni".pauza,
                        PT := T#10s,
                        ET => "Avarii".timer_eticheta);
   "Aparate".plecat_ethicheta := "timer_eticheta".Q;
   IF "timer_eticheta".Q THEN "Aparate".ajuns_eticheta := FALSE; END_IF;
   "Banda".banda_oprita_3 := "Aparate".ajuns_eticheta;
END_REGION

REGION Network 22: seteaza ca a ajuns la impachetare
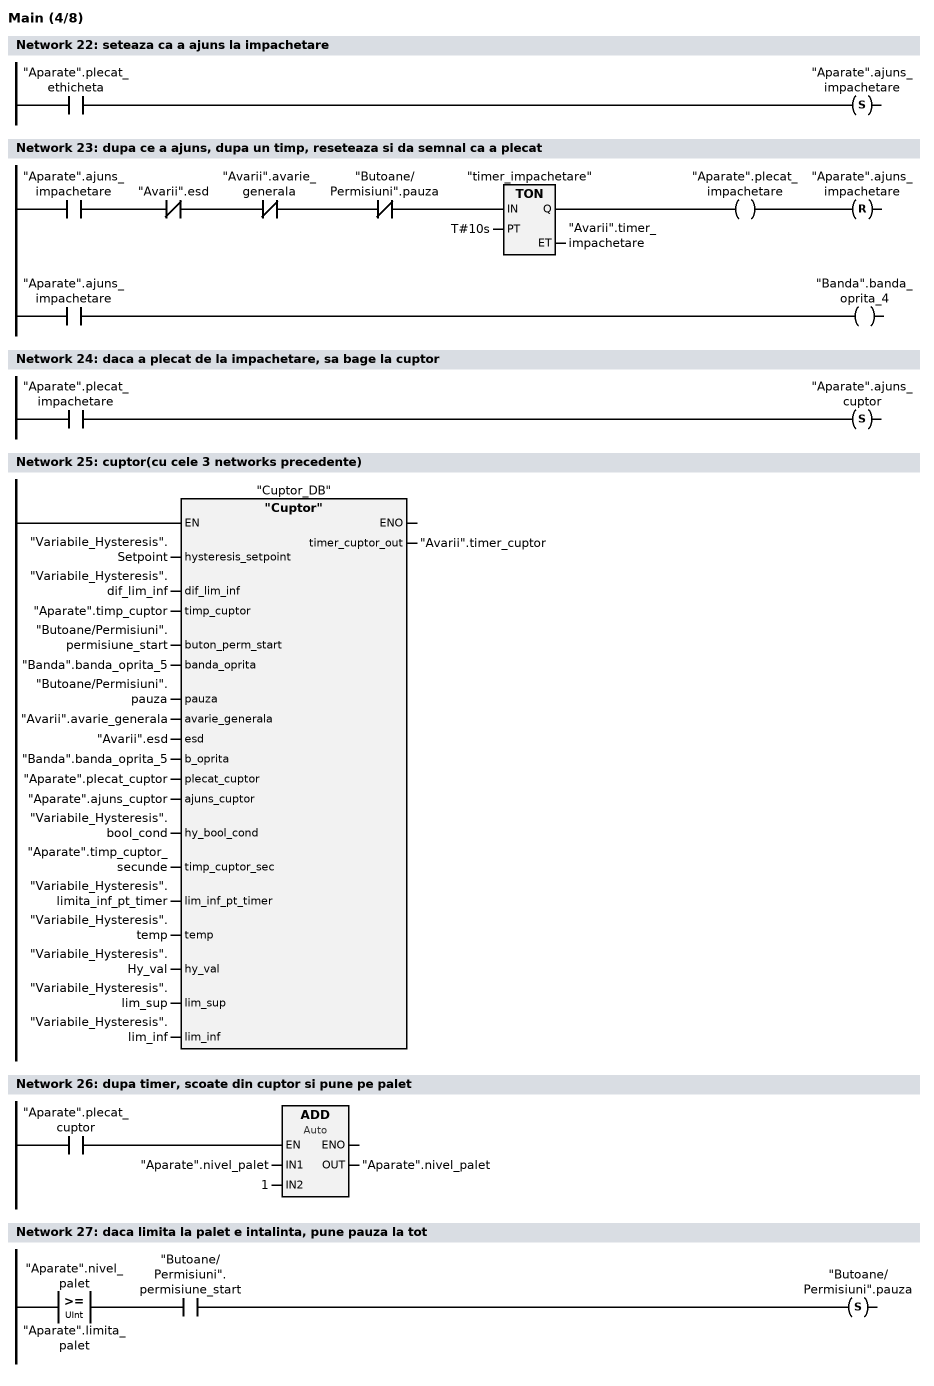
   RUNG wire#powerrail
      Contact( "Aparate".plecat_ethicheta )
      S_Coil( "Aparate".ajuns_impachetare )
   END_RUNG
   // the same network as SCL:
   IF "Aparate".plecat_ethicheta THEN "Aparate".ajuns_impachetare := TRUE; END_IF;
END_REGION

REGION Network 23: dupa ce a ajuns, dupa un timp, reseteaza si da semnal ca a plecat
   "timer_impachetare".TON(IN := "Aparate".ajuns_impachetare AND NOT "Avarii".esd AND NOT "Avarii".avarie_generala AND NOT "Butoane/Permisiuni".pauza,
                           PT := T#10s,
                           ET => "Avarii".timer_impachetare);
   "Aparate".plecat_impachetare := "timer_impachetare".Q;
   IF "timer_impachetare".Q THEN "Aparate".ajuns_impachetare := FALSE; END_IF;
   "Banda".banda_oprita_4 := "Aparate".ajuns_impachetare;
END_REGION

REGION Network 24: daca a plecat de la impachetare, sa bage la cuptor
   RUNG wire#powerrail
      Contact( "Aparate".plecat_impachetare )
      S_Coil( "Aparate".ajuns_cuptor )
   END_RUNG
   // the same network as SCL:
   IF "Aparate".plecat_impachetare THEN "Aparate".ajuns_cuptor := TRUE; END_IF;
END_REGION

REGION Network 25: cuptor(cu cele 3 networks precedente)
   RUNG wire#powerrail
      "Cuptor_DB"(hysteresis_setpoint := "Variabile_Hysteresis".Setpoint, dif_lim_inf := "Variabile_Hysteresis".dif_lim_inf, timp_cuptor := "Aparate".timp_cuptor, buton_perm_start := "Butoane/Permisiuni".permisiune_start, banda_oprita := "Banda".banda_oprita_5, pauza := "Butoane/Permisiuni".pauza, avarie_generala := "Avarii".avarie_generala, esd := "Avarii".esd, b_oprita := "Banda".banda_oprita_5, plecat_cuptor := "Aparate".plecat_cuptor, ajuns_cuptor := "Aparate".ajuns_cuptor, hy_bool_cond := "Variabile_Hysteresis".bool_cond, timp_cuptor_sec := "Aparate".timp_cuptor_secunde, lim_inf_pt_timer := "Variabile_Hysteresis".limita_inf_pt_timer, temp := "Variabile_Hysteresis".temp, hy_val := "Variabile_Hysteresis".Hy_val, lim_sup := "Variabile_Hysteresis".lim_sup, lim_inf := "Variabile_Hysteresis".lim_inf, timer_cuptor_out => "Avarii".timer_cuptor)
   END_RUNG
   // the same network as SCL:
   "Cuptor_DB"(hysteresis_setpoint := "Variabile_Hysteresis".Setpoint,   // "Cuptor"
               dif_lim_inf := "Variabile_Hysteresis".dif_lim_inf,
               timp_cuptor := "Aparate".timp_cuptor,
               buton_perm_start := "Butoane/Permisiuni".permisiune_start,
               banda_oprita := "Banda".banda_oprita_5,
               pauza := "Butoane/Permisiuni".pauza,
               avarie_generala := "Avarii".avarie_generala,
               esd := "Avarii".esd,
               b_oprita := "Banda".banda_oprita_5,
               plecat_cuptor := "Aparate".plecat_cuptor,
               ajuns_cuptor := "Aparate".ajuns_cuptor,
               hy_bool_cond := "Variabile_Hysteresis".bool_cond,
               timp_cuptor_sec := "Aparate".timp_cuptor_secunde,
               lim_inf_pt_timer := "Variabile_Hysteresis".limita_inf_pt_timer,
               temp := "Variabile_Hysteresis".temp,
               hy_val := "Variabile_Hysteresis".Hy_val,
               lim_sup := "Variabile_Hysteresis".lim_sup,
               lim_inf := "Variabile_Hysteresis".lim_inf,
               timer_cuptor_out => "Avarii".timer_cuptor);
END_REGION

REGION Network 26: dupa timer, scoate din cuptor si pune pe palet
   RUNG wire#powerrail
      Contact( "Aparate".plecat_cuptor )
      Add(in1 := "Aparate".nivel_palet, in2 := 1, out => "Aparate".nivel_palet)
   END_RUNG
   // the same network as SCL:
   IF "Aparate".plecat_cuptor THEN "Aparate".nivel_palet := "Aparate".nivel_palet + 1; END_IF;
END_REGION

REGION Network 27: daca limita la palet e intalinta, pune pauza la tot
   RUNG wire#powerrail
      { S7_Templates := "SrcType := UInt" } GE_Contact(in1 := "Aparate".nivel_palet, in2 := "Aparate".limita_palet)
      Contact( "Butoane/Permisiuni".permisiune_start )
      S_Coil( "Butoane/Permisiuni".pauza )
   END_RUNG
   // the same network as SCL:
   IF ("Aparate".nivel_palet >= "Aparate".limita_palet) AND "Butoane/Permisiuni".permisiune_start THEN
       "Butoane/Permisiuni".pauza := TRUE;
   END_IF;
END_REGION

REGION Network 28: simuleaza aici turnul vizual RGV
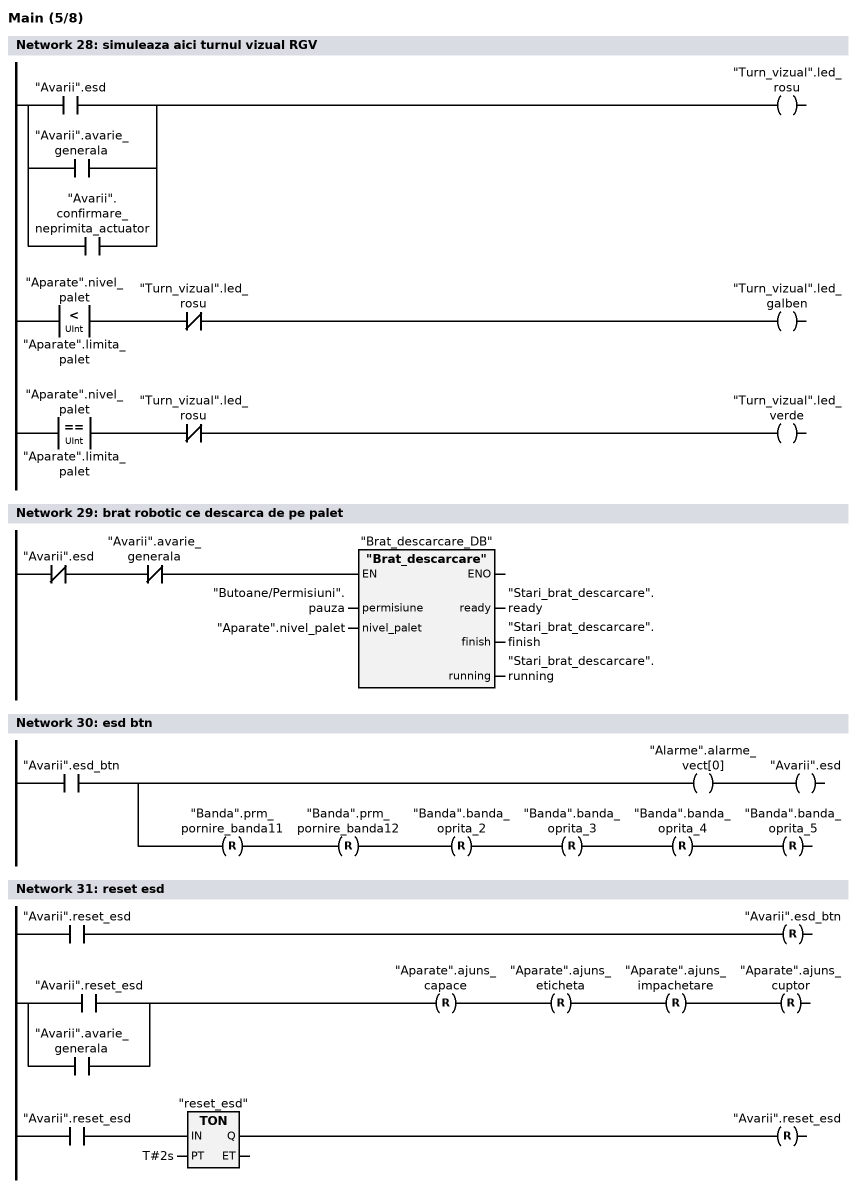
   RUNG wire#powerrail
      Contact( "Avarii".esd )
      wire#w1
      Coil( "Turn_vizual".led_rosu )
   END_RUNG
   RUNG wire#powerrail
      Contact( "Avarii".avarie_generala )
   END_RUNG wire#w1
   RUNG wire#powerrail
      Contact( "Avarii".confirmare_neprimita_actuator )
   END_RUNG wire#w1
   RUNG wire#powerrail
      { S7_Templates := "SrcType := UInt" } LT_Contact(in1 := "Aparate".nivel_palet, in2 := "Aparate".limita_palet)
      I_Contact( "Turn_vizual".led_rosu )
      Coil( "Turn_vizual".led_galben )
   END_RUNG
   RUNG wire#powerrail
      { S7_Templates := "SrcType := UInt" } EQ_Contact(in1 := "Aparate".nivel_palet, in2 := "Aparate".limita_palet)
      I_Contact( "Turn_vizual".led_rosu )
      Coil( "Turn_vizual".led_verde )
   END_RUNG
   // the same network as SCL:
   "Turn_vizual".led_rosu := "Avarii".esd OR "Avarii".avarie_generala OR "Avarii".confirmare_neprimita_actuator;
   "Turn_vizual".led_galben := ("Aparate".nivel_palet < "Aparate".limita_palet) AND NOT "Turn_vizual".led_rosu;
   "Turn_vizual".led_verde := ("Aparate".nivel_palet = "Aparate".limita_palet) AND NOT "Turn_vizual".led_rosu;
END_REGION

REGION Network 29: brat robotic ce descarca de pe palet
   RUNG wire#powerrail
      I_Contact( "Avarii".esd )
      I_Contact( "Avarii".avarie_generala )
      "Brat_descarcare_DB"(permisiune := "Butoane/Permisiuni".pauza, nivel_palet := "Aparate".nivel_palet, ready => "Stari_brat_descarcare".ready, finish => "Stari_brat_descarcare".finish, running => "Stari_brat_descarcare".running)
   END_RUNG
   // the same network as SCL:
   IF NOT "Avarii".esd AND NOT "Avarii".avarie_generala THEN
       "Brat_descarcare_DB"(permisiune := "Butoane/Permisiuni".pauza,   // "Brat_descarcare"
                            nivel_palet := "Aparate".nivel_palet,
                            ready => "Stari_brat_descarcare".ready,
                            finish => "Stari_brat_descarcare".finish,
                            running => "Stari_brat_descarcare".running);
   END_IF;
END_REGION

REGION Network 30: esd btn
   RUNG wire#powerrail
      Contact( "Avarii".esd_btn )
      wire#w1
      Coil( "Alarme".alarme_vect[0] )
      Coil( "Avarii".esd )
   END_RUNG
   RUNG wire#w1
      R_Coil( "Banda".prm_pornire_banda11 )
      R_Coil( "Banda".prm_pornire_banda12 )
      R_Coil( "Banda".banda_oprita_2 )
      R_Coil( "Banda".banda_oprita_3 )
      R_Coil( "Banda".banda_oprita_4 )
      R_Coil( "Banda".banda_oprita_5 )
   END_RUNG
   // the same network as SCL:
   "Alarme".alarme_vect[0] := "Avarii".esd_btn;
   "Avarii".esd := "Avarii".esd_btn;
   IF "Avarii".esd_btn THEN
       "Banda".prm_pornire_banda11 := FALSE;
       "Banda".prm_pornire_banda12 := FALSE;
       "Banda".banda_oprita_2 := FALSE;
       "Banda".banda_oprita_3 := FALSE;
       "Banda".banda_oprita_4 := FALSE;
       "Banda".banda_oprita_5 := FALSE;
   END_IF;
END_REGION

REGION Network 31: reset esd
   IF "Avarii".reset_esd THEN "Avarii".esd_btn := FALSE; END_IF;
   IF "Avarii".reset_esd OR "Avarii".avarie_generala THEN
       "Aparate".ajuns_capace := FALSE;
       "Aparate".ajuns_eticheta := FALSE;
       "Aparate".ajuns_impachetare := FALSE;
       "Aparate".ajuns_cuptor := FALSE;
   END_IF;
   "reset_esd".TON(IN := "Avarii".reset_esd, PT := T#2s);
   IF "reset_esd".Q THEN "Avarii".reset_esd := FALSE; END_IF;
END_REGION

REGION Network 32: avarie generala provocata de o avarie la unul din aparate
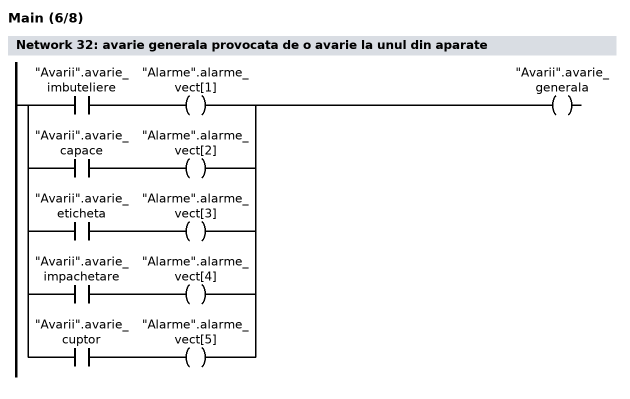
   RUNG wire#powerrail
      Contact( "Avarii".avarie_imbuteliere )
      Coil( "Alarme".alarme_vect[1] )
      wire#w1
      Coil( "Avarii".avarie_generala )
   END_RUNG
   RUNG wire#powerrail
      Contact( "Avarii".avarie_capace )
      Coil( "Alarme".alarme_vect[2] )
   END_RUNG wire#w1
   RUNG wire#powerrail
      Contact( "Avarii".avarie_eticheta )
      Coil( "Alarme".alarme_vect[3] )
   END_RUNG wire#w1
   RUNG wire#powerrail
      Contact( "Avarii".avarie_impachetare )
      Coil( "Alarme".alarme_vect[4] )
   END_RUNG wire#w1
   RUNG wire#powerrail
      Contact( "Avarii".avarie_cuptor )
      Coil( "Alarme".alarme_vect[5] )
   END_RUNG wire#w1
   // the same network as SCL:
   "Alarme".alarme_vect[1] := "Avarii".avarie_imbuteliere;
   "Alarme".alarme_vect[2] := "Avarii".avarie_capace;
   "Alarme".alarme_vect[3] := "Avarii".avarie_eticheta;
   "Alarme".alarme_vect[4] := "Avarii".avarie_impachetare;
   "Alarme".alarme_vect[5] := "Avarii".avarie_cuptor;
   "Avarii".avarie_generala := "Avarii".avarie_imbuteliere OR "Avarii".avarie_capace OR "Avarii".avarie_eticheta OR "Avarii".avarie_impachetare OR "Avarii".avarie_cuptor;
END_REGION

REGION Network 33: setare alarme hmi
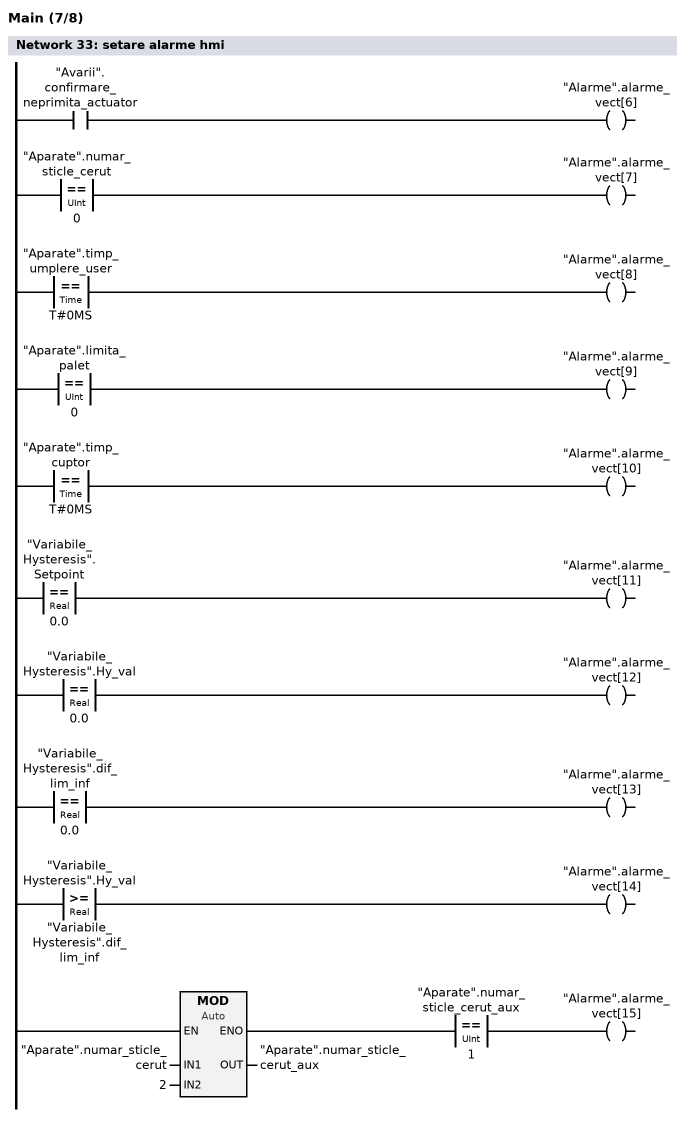
   RUNG wire#powerrail
      Contact( "Avarii".confirmare_neprimita_actuator )
      Coil( "Alarme".alarme_vect[6] )
   END_RUNG
   RUNG wire#powerrail
      { S7_Templates := "SrcType := UInt" } EQ_Contact(in1 := "Aparate".numar_sticle_cerut, in2 := 0)
      Coil( "Alarme".alarme_vect[7] )
   END_RUNG
   RUNG wire#powerrail
      { S7_Templates := "SrcType := Time" } EQ_Contact(in1 := "Aparate".timp_umplere_user, in2 := T#0MS)
      Coil( "Alarme".alarme_vect[8] )
   END_RUNG
   RUNG wire#powerrail
      { S7_Templates := "SrcType := UInt" } EQ_Contact(in1 := "Aparate".limita_palet, in2 := 0)
      Coil( "Alarme".alarme_vect[9] )
   END_RUNG
   RUNG wire#powerrail
      { S7_Templates := "SrcType := Time" } EQ_Contact(in1 := "Aparate".timp_cuptor, in2 := T#0MS)
      Coil( "Alarme".alarme_vect[10] )
   END_RUNG
   RUNG wire#powerrail
      { S7_Templates := "SrcType := Real" } EQ_Contact(in1 := "Variabile_Hysteresis".Setpoint, in2 := 0.0)
      Coil( "Alarme".alarme_vect[11] )
   END_RUNG
   RUNG wire#powerrail
      { S7_Templates := "SrcType := Real" } EQ_Contact(in1 := "Variabile_Hysteresis".Hy_val, in2 := 0.0)
      Coil( "Alarme".alarme_vect[12] )
   END_RUNG
   RUNG wire#powerrail
      { S7_Templates := "SrcType := Real" } EQ_Contact(in1 := "Variabile_Hysteresis".dif_lim_inf, in2 := 0.0)
      Coil( "Alarme".alarme_vect[13] )
   END_RUNG
   RUNG wire#powerrail
      { S7_Templates := "SrcType := Real" } GE_Contact(in1 := "Variabile_Hysteresis".Hy_val, in2 := "Variabile_Hysteresis".dif_lim_inf)
      Coil( "Alarme".alarme_vect[14] )
   END_RUNG
   RUNG wire#powerrail
      Mod(in1 := "Aparate".numar_sticle_cerut, in2 := 2, out => "Aparate".numar_sticle_cerut_aux)
      { S7_Templates := "SrcType := UInt" } EQ_Contact(in1 := "Aparate".numar_sticle_cerut_aux, in2 := 1)
      Coil( "Alarme".alarme_vect[15] )
   END_RUNG
   // the same network as SCL:
   "Alarme".alarme_vect[6] := "Avarii".confirmare_neprimita_actuator;
   "Alarme".alarme_vect[7] := "Aparate".numar_sticle_cerut = 0;
   "Alarme".alarme_vect[8] := "Aparate".timp_umplere_user = T#0MS;
   "Alarme".alarme_vect[9] := "Aparate".limita_palet = 0;
   "Alarme".alarme_vect[10] := "Aparate".timp_cuptor = T#0MS;
   "Alarme".alarme_vect[11] := "Variabile_Hysteresis".Setpoint = 0.0;
   "Alarme".alarme_vect[12] := "Variabile_Hysteresis".Hy_val = 0.0;
   "Alarme".alarme_vect[13] := "Variabile_Hysteresis".dif_lim_inf = 0.0;
   "Alarme".alarme_vect[14] := "Variabile_Hysteresis".Hy_val >= "Variabile_Hysteresis".dif_lim_inf;
   "Aparate".numar_sticle_cerut_aux := "Aparate".numar_sticle_cerut MOD 2;
   "Alarme".alarme_vect[15] := "Aparate".numar_sticle_cerut_aux = 1;
END_REGION

REGION Network 34: timp in secunde pt simulare (pe hmi)
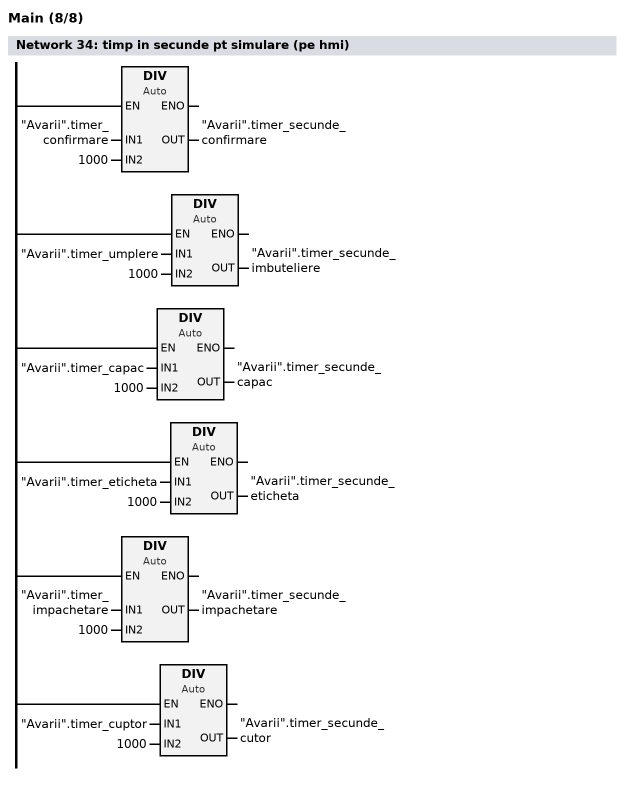
   RUNG wire#powerrail
      Div(in1 := "Avarii".timer_confirmare, in2 := 1000, out => "Avarii".timer_secunde_confirmare)
   END_RUNG
   RUNG wire#powerrail
      Div(in1 := "Avarii".timer_umplere, in2 := 1000, out => "Avarii".timer_secunde_imbuteliere)
   END_RUNG
   RUNG wire#powerrail
      Div(in1 := "Avarii".timer_capac, in2 := 1000, out => "Avarii".timer_secunde_capac)
   END_RUNG
   RUNG wire#powerrail
      Div(in1 := "Avarii".timer_eticheta, in2 := 1000, out => "Avarii".timer_secunde_eticheta)
   END_RUNG
   RUNG wire#powerrail
      Div(in1 := "Avarii".timer_impachetare, in2 := 1000, out => "Avarii".timer_secunde_impachetare)
   END_RUNG
   RUNG wire#powerrail
      Div(in1 := "Avarii".timer_cuptor, in2 := 1000, out => "Avarii".timer_secunde_cutor)
   END_RUNG
   // the same network as SCL:
   "Avarii".timer_secunde_confirmare := "Avarii".timer_confirmare / 1000;
   "Avarii".timer_secunde_imbuteliere := "Avarii".timer_umplere / 1000;
   "Avarii".timer_secunde_capac := "Avarii".timer_capac / 1000;
   "Avarii".timer_secunde_eticheta := "Avarii".timer_eticheta / 1000;
   "Avarii".timer_secunde_impachetare := "Avarii".timer_impachetare / 1000;
   "Avarii".timer_secunde_cutor := "Avarii".timer_cuptor / 1000;
END_REGION
END_ORGANIZATION_BLOCK

(* ===== HMI "HMI_RT_1" =====
system functions are stored by id; their names below are inferred from use
connection "HMI_Connection_1": ETHERNET, SMART_S7_1500_OMS

HMI tags "Default tag table"
   "Tag_ScreenNumber" : UInt, internal
   "Variabile_Hysteresis_temp" : Real = PLC Variabile_Hysteresis.temp, 1 s
   "Aparate_numar_sticle_cerut" : UInt = PLC Aparate.numar_sticle_cerut, 1 s
   "Aparate_limita_palet" : UInt = PLC Aparate.limita_palet, 1 s
   "Aparate_timp_cuptor" : Time = PLC Aparate.timp_cuptor, 1 s
   "Aparate_timp_umplere_user" : Time = PLC Aparate.timp_umplere_user, 1 s
   "Variabile_Hysteresis_Setpoint" : Real = PLC Variabile_Hysteresis.Setpoint, 1 s
   "Variabile_Hysteresis_Hy_val" : Real = PLC Variabile_Hysteresis.Hy_val, 1 s
   "Avarii_esd" : Bool = PLC Avarii.esd, 1 s
   "Avarii_esd_btn" : Bool = PLC Avarii.esd_btn, 1 s
   "Avarii_reset_esd" : Bool = PLC Avarii.reset_esd, 1 s
   "Avarii_confirmare_neprimita_actuator" : Bool = PLC Avarii.confirmare_neprimita_actuator, 1 s
   "Avarii_avarie_imbuteliere" : Bool = PLC Avarii.avarie_imbuteliere, 1 s
   "Avarii_avarie_capace" : Bool = PLC Avarii.avarie_capace, 1 s
   "Avarii_avarie_eticheta" : Bool = PLC Avarii.avarie_eticheta, 1 s
   "Avarii_avarie_impachetare" : Bool = PLC Avarii.avarie_impachetare, 1 s
   "Avarii_avarie_cuptor" : Bool = PLC Avarii.avarie_cuptor, 1 s
   "Avarii_reset_avarii" : Bool = PLC Avarii.reset_avarii, 1 s
   "Aparate_confirmare_actuator" : Bool = PLC Aparate.confirmare_actuator, 1 s
   "Avarii_timer_confirmare" : Time = PLC Avarii.timer_confirmare, 1 s
   "Avarii_var_confirmare" : Bool = PLC Avarii.var_confirmare, 1 s
   "Aparate_nivel_palet" : UInt = PLC Aparate.nivel_palet, 1 s
   "Stari_brat_descarcare_ready" : Bool = PLC Stari_brat_descarcare.ready, 1 s
   "Stari_brat_descarcare_finish" : Bool = PLC Stari_brat_descarcare.finish, 1 s
   "Stari_brat_descarcare_running" : Bool = PLC Stari_brat_descarcare.running, 1 s
   "Turn_vizual_led_rosu" : Bool = PLC Turn_vizual.led_rosu, 1 s
   "Turn_vizual_led_galben" : Bool = PLC Turn_vizual.led_galben, 1 s
   "Turn_vizual_led_verde" : Bool = PLC Turn_vizual.led_verde, 1 s
   "Butoane/Permisiuni_btn_start" : Bool = PLC "Butoane/Permisiuni".btn_start, 1 s
   "Butoane/Permisiuni_pauza" : Bool = PLC "Butoane/Permisiuni".pauza, 1 s
   "Alarme_alarme_gather" : Word = PLC Alarme.alarme_gather, 1 s
   "Banda_banda_pornita_1" : Bool = PLC Banda.banda_pornita_1, 1 s
   "Banda_banda_oprita_2" : Bool = PLC Banda.banda_oprita_2, 1 s
   "Banda_banda_oprita_3" : Bool = PLC Banda.banda_oprita_3, 1 s
   "Banda_banda_oprita_4" : Bool = PLC Banda.banda_oprita_4, 1 s
   "Banda_banda_oprita_5" : Bool = PLC Banda.banda_oprita_5, 1 s
   "Aparate_numar_sticle" : UInt = PLC Aparate.numar_sticle, 1 s
   "Avarii_timer_umplere" : Time = PLC Avarii.timer_umplere, 1 s
   "Aparate_inchidere_actuator" : Bool = PLC Aparate.inchidere_actuator, 1 s
   "Avarii_timer_capac" : Time = PLC Avarii.timer_capac, 1 s
   "Aparate_ajuns_capace" : Bool = PLC Aparate.ajuns_capace, 1 s
   "Aparate_ajuns_eticheta" : Bool = PLC Aparate.ajuns_eticheta, 1 s
   "Avarii_timer_eticheta" : Time = PLC Avarii.timer_eticheta, 1 s
   "Avarii_timer_impachetare" : Time = PLC Avarii.timer_impachetare, 1 s
   "Aparate_ajuns_impachetare" : Bool = PLC Aparate.ajuns_impachetare, 1 s
   "Aparate_ajuns_cuptor" : Bool = PLC Aparate.ajuns_cuptor, 1 s
   "Avarii_timer_secunde_confirmare" : Time = PLC Avarii.timer_secunde_confirmare, 1 s
   "Avarii_timer_secunde_imbuteliere" : Time = PLC Avarii.timer_secunde_imbuteliere, 1 s
   "Avarii_timer_secunde_capac" : Time = PLC Avarii.timer_secunde_capac, 1 s
   "Avarii__timer_secunde_eticheta" : Time = PLC Avarii.timer_secunde_eticheta, 1 s
   "Avarii_timer_secunde_impachetare" : Time = PLC Avarii.timer_secunde_impachetare, 1 s
   "Avarii_timer_secunde_cutor" : Time = PLC Avarii.timer_secunde_cutor, 1 s
   "Variabile_Hysteresis_dif_lim_inf" : Real = PLC Variabile_Hysteresis.dif_lim_inf, 1 s

discrete alarms
   1: 'ESD', class Errors, trigger "Alarme_alarme_gather" bit 0
   2: 'Avarie imbuteliere', class Errors, trigger "Alarme_alarme_gather" bit 1
   3: 'Avarie capace', class Errors, trigger "Alarme_alarme_gather" bit 2
   4: 'Avarie eticheta', class Errors, trigger "Alarme_alarme_gather" bit 3
   5: 'Avarie impachetare', class Errors, trigger "Alarme_alarme_gather" bit 4
   6: 'Avarie cuptor', class Errors, trigger "Alarme_alarme_gather" bit 5
   7: 'Confirmare naprimita', class Errors, trigger "Alarme_alarme_gather" bit 6
   8: 'Numar sticle neintrodus', class Errors, trigger "Alarme_alarme_gather" bit 7
   9: 'Timp umplere neintrodus', class Errors, trigger "Alarme_alarme_gather" bit 8
   10: 'Limita palet neintrodusa', class Errors, trigger "Alarme_alarme_gather" bit 9
   11: 'Timp cuptor neintrodus', class Errors, trigger "Alarme_alarme_gather" bit 10
   12: 'Temperatura cuptor neintrodusa', class Errors, trigger "Alarme_alarme_gather" bit 11
   13: 'Valoare hysteresis neintrodusa', class Errors, trigger "Alarme_alarme_gather" bit 12
   14: 'Limita inf. pt calcul simulare neintrodusa', class Errors, trigger "Alarme_alarme_gather" bit 13
   15: 'Valoarea depaseste limita de calcul', class Errors, trigger "Alarme_alarme_gather" bit 14
   16: 'Limita de sticle trebuie sa fie un numar par', class Errors, trigger "Alarme_alarme_gather" bit 15

Template "Template_1" 800x480
   Button "Exit" at 722,440 size 55x39; TextOff 'Exit'; PictureOff "ExitRuntime_KTP900_Basic_PN_TR"; PictureOn "ExitRuntime_KTP900_Basic_PN_TR"
      on Release: StopRuntime(0)
   Button "Template_Button" at 622,440 size 55x39; TextOff 'Text'
   Button "Template_Button_1" at 522,440 size 55x39; TextOff 'Text'
   Button "Alarms" at 622,440 size 55x39; TextOff 'Alarms'; PictureOff "AlarmDisplay_KTP900_Basic_PN_TR"; PictureOn "AlarmDisplay_KTP900_Basic_PN_TR"
      on Release: function_ef3f5d25("Alarm window_1", -1)
   Button "Start screen" at 522,440 size 55x39; TextOff 'Start screen'; PictureOff "NavigateHome_KTP900_Basic_PN_TR"; PictureOn "NavigateHome_KTP900_Basic_PN_TR"
      on Release: ActivateScreen("Main", 0)
   SymbolicIOField "Symbolic_IO_Field_Screen" at 73,7 size 620x26; TextOff '0'; TextOn '1'; TextList "TextList_ScreenNames"
      ProcessValue <- "Tag_ScreenNumber"
      on Change: ActivateScreenByNumber("Tag_ScreenNumber", 0)
   DateTimeField "HmiScreenItemData" at 695,20 size 105x20
   DateTimeField "HmiScreenItemData_1" at 695,0 size 105x20
   GraphicView "Logo" at 0,0 size 71x40; Picture "Logo of HMI_1"

screen "Main" 800x480, template "Template_1"
   on GenerateScreen: SetTag("Tag_ScreenNumber", 1)
   TextField "Text field_1" at 31,460 size 35x20; Text 'Main'
   TextField "Text field_2" at 119,460 size 60x20; Text 'Simulare'
   TextField "Text field_3" at 231,460 size 42x20; Text 'Grafic'
   TextField "Text field_4" at 359,6 size 46x25; Text 'Main'
   TextField "Text field_5" at 665,50 size 43x20; Text 'Avarii'
   Button "Button_1" at 370,387 size 55x32; TextOff 'ESD'
      on Click: SetBit("Avarii_esd_btn")
   Button "Button_2" at 370,428 size 55x32; TextOff 'RESET'
      on Click: SetBit("Avarii_reset_esd")
   Circle "Circle_1" at 374,327 size 48x48
      Appearance <- "Avarii_esd"
   IOField "I/O field_1" at 46,131 size 96x32; FormatPattern 999
      ProcessValue <- "Aparate_numar_sticle_cerut"
   TextField "Text field_6" at 46,107 size 84x20; Text 'Numar sticle'
   IOField "I/O field_2" at 46,199 size 96x32; FormatPattern 999
      ProcessValue <- "Aparate_limita_palet"
   TextField "Text field_7" at 46,175 size 80x20; Text 'Limita palet'
   IOField "I/O field_3" at 46,267 size 96x32; FormatPattern 9999
      ProcessValue <- "Variabile_Hysteresis_Setpoint"
   TextField "Text field_8" at 46,243 size 89x20; Text 'Temperatura'
   IOField "I/O field_4" at 179,131 size 96x32; FormatPattern 9999; Unit s
      ProcessValue <- "Aparate_timp_umplere_user"
   TextField "Text field_9" at 179,107 size 90x20; Text 'Timp umplere'
   IOField "I/O field_5" at 177,198 size 96x32; FormatPattern 9999; Unit s
      ProcessValue <- "Aparate_timp_cuptor"
   TextField "Text field_10" at 177,174 size 81x20; Text 'Timp cuptor'
   IOField "I/O field_6" at 175,265 size 96x32; FormatPattern 999.9
      ProcessValue <- "Variabile_Hysteresis_dif_lim_inf"
   TextField "Text field_11" at 175,241 size 50x20; Text 'Lim_inf'
   Button "Button_3" at 646,371 size 96x32; TextOff 'RESET'
      on Click: SetBit("Avarii_reset_avarii")
   Circle "Circle_2" at 633,77 size 31x31
      Appearance <- "Avarii_confirmare_neprimita_actuator"
   TextField "Text field_12" at 671,77 size 80x20; Text 'Confirmare'
   TextField "Text field_13" at 678,94 size 66x20; Text 'neprimita'
   Button "Button_4" at 678,125 size 96x32; TextOff 'Imbuteliere'
      on Click: SetBit("Avarii_avarie_imbuteliere")
   Circle "Circle_3" at 633,124 size 31x31
      Appearance <- "Avarii_avarie_imbuteliere"
   Circle "Circle_4" at 633,171 size 31x31
      Appearance <- "Avarii_avarie_capace"
   Circle "Circle_5" at 633,218 size 31x31
      Appearance <- "Avarii_avarie_eticheta"
   Circle "Circle_6" at 633,265 size 31x31
      Appearance <- "Avarii_avarie_impachetare"
   Circle "Circle_7" at 633,312 size 31x31
      Appearance <- "Avarii_avarie_cuptor"
   Button "Button_5" at 678,171 size 96x32; TextOff 'Capace'
      on Click: SetBit("Avarii_avarie_capace")
   Button "Button_6" at 678,217 size 96x32; TextOff 'Eticheta'
      on Click: SetBit("Avarii_avarie_eticheta")
   Button "Button_7" at 678,263 size 96x32; TextOff 'Impachetare'
      on Click: SetBit("Avarii_avarie_impachetare")
   Button "Button_8" at 678,309 size 96x32; TextOff 'Cuptor'
      on Click: SetBit("Avarii_avarie_cuptor")
   IOField "I/O field_7" at 310,65 size 96x32; FormatPattern 99; Unit s
      Visibility <- "Avarii_var_confirmare"
      ProcessValue <- "Avarii_timer_secunde_confirmare"
   Button "Button_9" at 416,65 size 61x32; TextOff 'Confirm'
      on Click: SetBit("Aparate_confirmare_actuator")
      Visibility <- "Avarii_var_confirmare"
   TextField "Text field_14" at 338,45 size 115x20; Text 'Timer Confirmare'
      Visibility <- "Avarii_var_confirmare"
   IOField "I/O field_8" at 176,329 size 96x32; FormatPattern 999.9
      ProcessValue <- "Variabile_Hysteresis_Hy_val"
   TextField "Text field_15" at 176,305 size 142x20; Text 'Hysteresis(<Lim_inf)'

screen "Simulare" 800x480
   TextField "Text field_1" at 31,460 size 35x20; Text 'Main'
   TextField "Text field_2" at 119,460 size 60x20; Text 'Simulare'
   TextField "Text field_3" at 231,460 size 42x20; Text 'Grafic'
   TextField "Text field_4" at 355,3 size 80x25; Text 'Simulare'
   Rectangle "Rectangle_1" at 92,239 size 102x24
      Appearance <- "Banda_banda_pornita_1"
   Rectangle "Rectangle_2" at 210,239 size 102x24
      Appearance <- "Banda_banda_oprita_2"
   Rectangle "Rectangle_3" at 322,239 size 102x24
      Appearance <- "Banda_banda_oprita_3"
   Rectangle "Rectangle_4" at 433,239 size 102x24
      Appearance <- "Banda_banda_oprita_4"
   Rectangle "Rectangle_5" at 544,239 size 102x24
      Appearance <- "Banda_banda_oprita_5"
   Button "Button_1" at 14,235 size 52x32; TextOff 'Start'
      on Click: SetBit("Butoane/Permisiuni_btn_start")
   Circle "Circle_1" at 461,347 size 29x29
      Appearance <- "Turn_vizual_led_rosu"
   Circle "Circle_2" at 461,376 size 29x29
      Appearance <- "Turn_vizual_led_galben"
   Circle "Circle_3" at 461,405 size 29x29
      Appearance <- "Turn_vizual_led_verde"
   TextField "Text field_5" at 425,323 size 106x20; Text 'Indicator Vizual'
   IOField "I/O field_1" at 651,33 size 96x32; FormatPattern 9999
      ProcessValue <- "Aparate_nivel_palet"
   Circle "Circle_4" at 729,185 size 29x29
      Appearance <- "Stari_brat_descarcare_ready"
   Circle "Circle_5" at 729,214 size 29x29
      Appearance <- "Stari_brat_descarcare_running"
   Circle "Circle_6" at 729,243 size 29x29
      Appearance <- "Stari_brat_descarcare_finish"
   TextField "Text field_6" at 689,161 size 110x20; Text 'Brat descarcare'
   TextField "Text field_7" at 689,187 size 30x20; Text 'Rdy'
   TextField "Text field_8" at 689,214 size 30x20; Text 'Run'
   TextField "Text field_9" at 692,243 size 22x20; Text 'Fin'
   TextField "Text field_10" at 642,12 size 103x20; Text 'Cantitate palet'
   Rectangle "Rectangle_6" at 111,187 size 59x35
      Appearance <- "Aparate_inchidere_actuator"
   Rectangle "Rectangle_7" at 245,156 size 29x65
      Appearance <- "Aparate_ajuns_capace"
   Rectangle "Rectangle_8" at 355,154 size 29x65
      Appearance <- "Aparate_ajuns_eticheta"
   Rectangle "Rectangle_9" at 465,155 size 29x65
      Appearance <- "Aparate_ajuns_impachetare"
   Rectangle "Rectangle_10" at 569,187 size 59x35
      Appearance <- "Aparate_ajuns_cuptor"
   IOField "I/O field_2" at 555,138 size 96x32; FormatPattern 9999.99
      ProcessValue <- "Variabile_Hysteresis_temp"
   TextField "Text field_11" at 556,118 size 89x20; Text 'Temperatura'
   IOField "I/O field_3" at 56,25 size 96x32; FormatPattern 99; Unit s
      Visibility <- "Avarii_var_confirmare"
      ProcessValue <- "Avarii_timer_secunde_confirmare"
   Button "Button_2" at 162,25 size 61x32; TextOff 'Confirm'
      on Click: SetBit("Aparate_confirmare_actuator")
      Visibility <- "Avarii_var_confirmare"
   TextField "Text field_12" at 84,5 size 115x20; Text 'Timer Confirmare'
      Visibility <- "Avarii_var_confirmare"
   IOField "I/O field_4" at 48,145 size 36x32; FormatPattern 999
      ProcessValue <- "Aparate_numar_sticle"
   TextField "Text field_13" at 46,125 size 40x20; Text 'Sticle'
   Circle "Circle_7" at 152,371 size 48x48
      Appearance <- "Butoane/Permisiuni_pauza"
   TextField "Text field_14" at 153,350 size 44x20; Text 'Pauza'
   IOField "I/O field_5" at 113,146 size 54x32; FormatPattern 99; Unit s
      ProcessValue <- "Avarii_timer_secunde_imbuteliere"
   TextField "Text field_15" at 112,125 size 57x20; Text 'Umplere'
   IOField "I/O field_6" at 231,113 size 54x32; FormatPattern 99; Unit s
      ProcessValue <- "Avarii_timer_secunde_capac"
   TextField "Text field_16" at 230,92 size 52x20; Text 'Capace'
   IOField "I/O field_7" at 344,112 size 54x32; FormatPattern 99; Unit s
      ProcessValue <- "Avarii__timer_secunde_eticheta"
   TextField "Text field_17" at 343,91 size 58x20; Text 'Eticheta'
   IOField "I/O field_8" at 453,114 size 54x32; FormatPattern 99; Unit s
      ProcessValue <- "Avarii_timer_secunde_impachetare"
   TextField "Text field_18" at 436,94 size 88x20; Text 'Impachetare'
   IOField "I/O field_9" at 569,79 size 54x32; FormatPattern 99; Unit s
      ProcessValue <- "Avarii_timer_secunde_cutor"
   TextField "Text field_19" at 568,58 size 49x20; Text 'Cuptor'
   TextField "Text field_20" at 493,350 size 48x20; Text 'Avarie'
   TextField "Text field_21" at 493,379 size 68x20; Text 'Incarcare'
   TextField "Text field_22" at 493,408 size 79x20; Text 'Descarcare'

screen "Temperatura_cuptor" 800x480
   TrendView "Trend view_1" at 26,62 size 739x375
   TextField "Text field_1" at 31,460 size 35x20; Text 'Main'
   TextField "Text field_2" at 119,460 size 60x20; Text 'Simulare'
   TextField "Text field_3" at 231,460 size 42x20; Text 'Grafic'
   TextField "Text field_4" at 310,16 size 177x25; Text 'Temperatura Cuptor'
   IOField "I/O field_3" at 56,25 size 96x32; FormatPattern 99; Unit s
      Visibility <- "Avarii_var_confirmare"
      ProcessValue <- "Avarii_timer_secunde_confirmare"
   Button "Button_2" at 162,25 size 61x32; TextOff 'Confirm'
      on Click: SetBit("Aparate_confirmare_actuator")
      Visibility <- "Avarii_var_confirmare"
   TextField "Text field_12" at 84,5 size 115x20; Text 'Timer Confirmare'
      Visibility <- "Avarii_var_confirmare"
*)